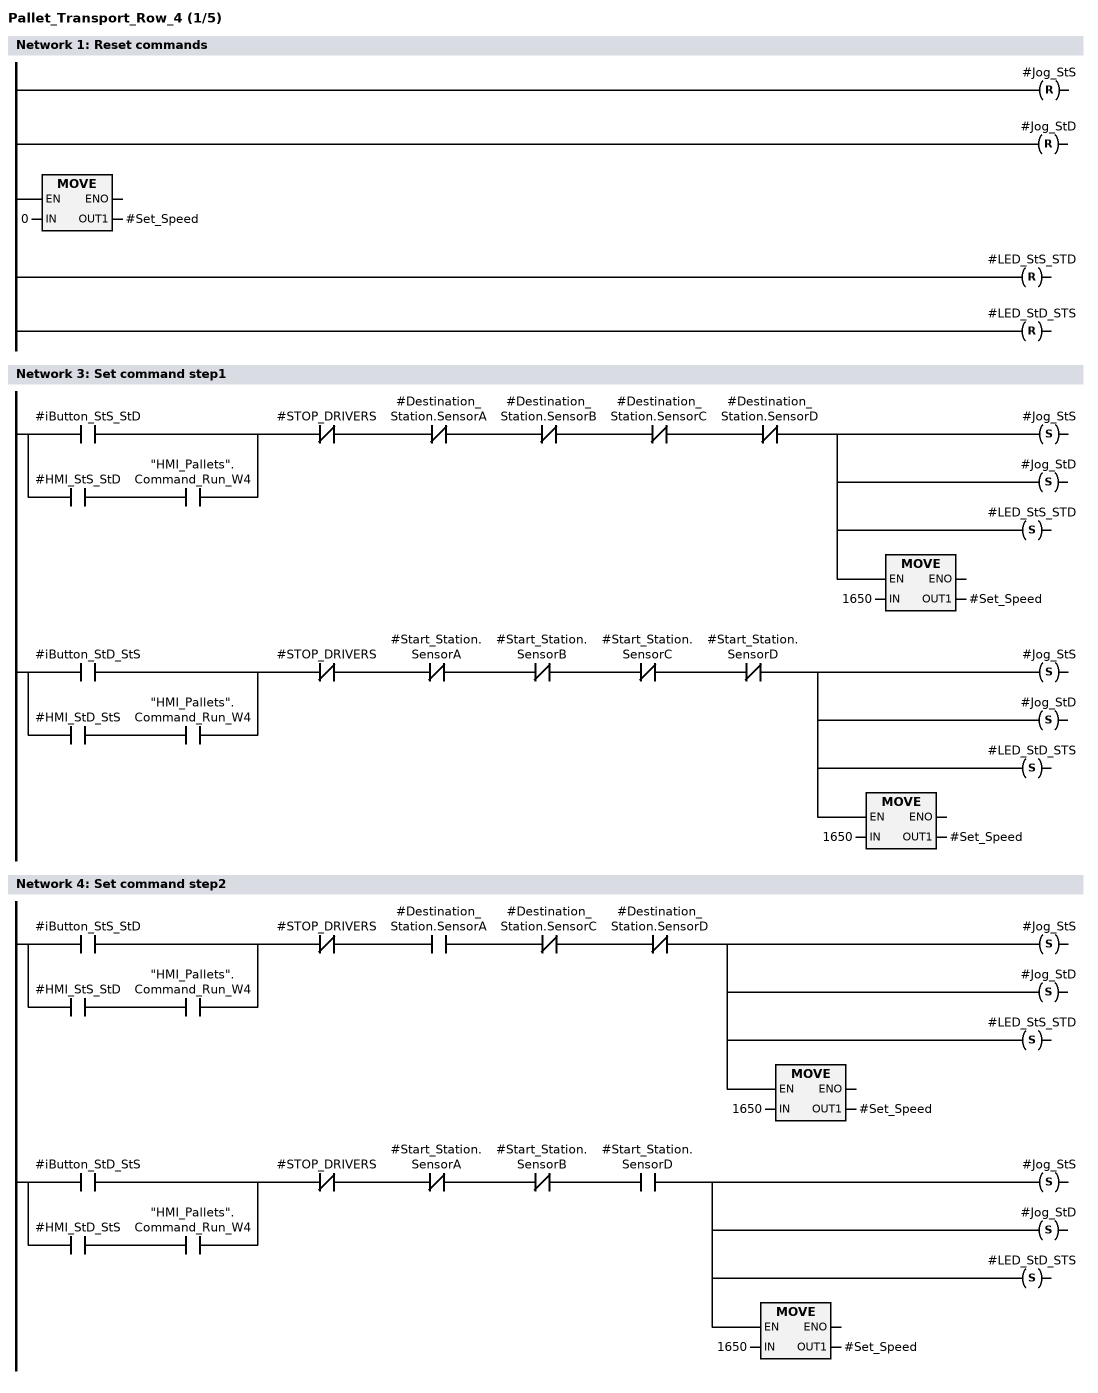
   RUNG wire#powerrail
      R_Coil( #Jog_StS )
   END_RUNG
   RUNG wire#powerrail
      R_Coil( #Jog_StD )
   END_RUNG
   RUNG wire#powerrail
      Move(in := 0, out1 => #Set_Speed)
   END_RUNG
   RUNG wire#powerrail
      R_Coil( #LED_StS_STD )
   END_RUNG
   RUNG wire#powerrail
      R_Coil( #LED_StD_STS )
   END_RUNG
   // the same network as SCL:
   #Jog_StS := FALSE;
   #Jog_StD := FALSE;
   #Set_Speed := 0;
   #LED_StS_STD := FALSE;
   #LED_StD_STS := FALSE;
END_REGION

REGION Network 2 (SCL): Triggers STOP_DRIVERS after 8 s of active move command without motion
   #Timer_Drive_Error_Button(
                             IN :=
                             (
                             #iButton_StS_StD OR
                             #iButton_StD_StS
                             )
                             AND NOT (
                             #oDriveStS_Param.x_Bit_4_Motor_turning OR
                             #oDriveStS_double_Param.x_Bit_4_Motor_turning OR
                             #oDriveStD_Param.x_Bit_4_Motor_turning OR
                             #oDriveStD_double_Param.x_Bit_4_Motor_turning
                             ),
                             PT := T#15s
   );


   #Timer_Drive_Error_HMI(
                          IN :=
                          (
                          #HMI_StS_StD OR
                          #HMI_StD_StS
                          )
                          AND NOT (
                          #oDriveStS_Param.x_Bit_4_Motor_turning OR
                          #oDriveStS_double_Param.x_Bit_4_Motor_turning OR
                          #oDriveStD_Param.x_Bit_4_Motor_turning OR
                          #oDriveStD_double_Param.x_Bit_4_Motor_turning
                          ),
                          PT := T#10s
   );

   IF #Timer_Drive_Error_Button.Q THEN
       #STOP_DRIVERS := TRUE;
       #Stop_Drive_Button := TRUE;
   END_IF;


   IF #Timer_Drive_Error_HMI.Q THEN
       #STOP_DRIVERS := TRUE;
       #Stop_Drive_HMI := TRUE;
       #HMI_StS_StD := FALSE;
       #HMI_StD_StS := FALSE;
   END_IF;


   IF "HMI_Pallets".Reset_Drivers THEN
       #STOP_DRIVERS := FALSE;
       #Stop_Drive_Button := FALSE;
       #Stop_Drive_HMI := FALSE;
   END_IF;
END_REGION

REGION Network 3: Set command step1
   RUNG wire#powerrail
      Contact( #iButton_StS_StD )
      wire#w1
      I_Contact( #STOP_DRIVERS )
      I_Contact( #Destination_Station.SensorA )
      I_Contact( #Destination_Station.SensorB )
      I_Contact( #Destination_Station.SensorC )
      I_Contact( #Destination_Station.SensorD )
      wire#w2
      S_Coil( #Jog_StS )
   END_RUNG
   RUNG wire#powerrail
      Contact( #HMI_StS_StD )
      Contact( "HMI_Pallets".Command_Run_W4 )
   END_RUNG wire#w1
   RUNG wire#w2
      S_Coil( #Jog_StD )
   END_RUNG
   RUNG wire#w2
      S_Coil( #LED_StS_STD )
   END_RUNG
   RUNG wire#w2
      Move(in := 1650, out1 => #Set_Speed)
   END_RUNG
   RUNG wire#powerrail
      Contact( #iButton_StD_StS )
      wire#w3
      I_Contact( #STOP_DRIVERS )
      I_Contact( #Start_Station.SensorA )
      I_Contact( #Start_Station.SensorB )
      I_Contact( #Start_Station.SensorC )
      I_Contact( #Start_Station.SensorD )
      wire#w4
      S_Coil( #Jog_StS )
   END_RUNG
   RUNG wire#powerrail
      Contact( #HMI_StD_StS )
      Contact( "HMI_Pallets".Command_Run_W4 )
   END_RUNG wire#w3
   RUNG wire#w4
      S_Coil( #Jog_StD )
   END_RUNG
   RUNG wire#w4
      S_Coil( #LED_StD_STS )
   END_RUNG
   RUNG wire#w4
      Move(in := 1650, out1 => #Set_Speed)
   END_RUNG
   // the same network as SCL:
   IF (#iButton_StS_StD OR (#HMI_StS_StD AND "HMI_Pallets".Command_Run_W4)) AND NOT #STOP_DRIVERS AND NOT #Destination_Station.SensorA AND NOT #Destination_Station.SensorB AND NOT #Destination_Station.SensorC AND NOT #Destination_Station.SensorD THEN
       #Jog_StS := TRUE;
       #Jog_StD := TRUE;
       #LED_StS_STD := TRUE;
       #Set_Speed := 1650;
   END_IF;
   IF (#iButton_StD_StS OR (#HMI_StD_StS AND "HMI_Pallets".Command_Run_W4)) AND NOT #STOP_DRIVERS AND NOT #Start_Station.SensorA AND NOT #Start_Station.SensorB AND NOT #Start_Station.SensorC AND NOT #Start_Station.SensorD THEN
       #Jog_StS := TRUE;
       #Jog_StD := TRUE;
       #LED_StD_STS := TRUE;
       #Set_Speed := 1650;
   END_IF;
END_REGION

REGION Network 4: Set command step2
   RUNG wire#powerrail
      Contact( #iButton_StS_StD )
      wire#w1
      I_Contact( #STOP_DRIVERS )
      Contact( #Destination_Station.SensorA )
      I_Contact( #Destination_Station.SensorC )
      I_Contact( #Destination_Station.SensorD )
      wire#w2
      S_Coil( #Jog_StS )
   END_RUNG
   RUNG wire#powerrail
      Contact( #HMI_StS_StD )
      Contact( "HMI_Pallets".Command_Run_W4 )
   END_RUNG wire#w1
   RUNG wire#w2
      S_Coil( #Jog_StD )
   END_RUNG
   RUNG wire#w2
      S_Coil( #LED_StS_STD )
   END_RUNG
   RUNG wire#w2
      Move(in := 1650, out1 => #Set_Speed)
   END_RUNG
   RUNG wire#powerrail
      Contact( #iButton_StD_StS )
      wire#w3
      I_Contact( #STOP_DRIVERS )
      I_Contact( #Start_Station.SensorA )
      I_Contact( #Start_Station.SensorB )
      Contact( #Start_Station.SensorD )
      wire#w4
      S_Coil( #Jog_StS )
   END_RUNG
   RUNG wire#powerrail
      Contact( #HMI_StD_StS )
      Contact( "HMI_Pallets".Command_Run_W4 )
   END_RUNG wire#w3
   RUNG wire#w4
      S_Coil( #Jog_StD )
   END_RUNG
   RUNG wire#w4
      S_Coil( #LED_StD_STS )
   END_RUNG
   RUNG wire#w4
      Move(in := 1650, out1 => #Set_Speed)
   END_RUNG
   // the same network as SCL:
   IF (#iButton_StS_StD OR (#HMI_StS_StD AND "HMI_Pallets".Command_Run_W4)) AND NOT #STOP_DRIVERS AND #Destination_Station.SensorA AND NOT #Destination_Station.SensorC AND NOT #Destination_Station.SensorD THEN
       #Jog_StS := TRUE;
       #Jog_StD := TRUE;
       #LED_StS_STD := TRUE;
       #Set_Speed := 1650;
   END_IF;
   IF (#iButton_StD_StS OR (#HMI_StD_StS AND "HMI_Pallets".Command_Run_W4)) AND NOT #STOP_DRIVERS AND NOT #Start_Station.SensorA AND NOT #Start_Station.SensorB AND #Start_Station.SensorD THEN
       #Jog_StS := TRUE;
       #Jog_StD := TRUE;
       #LED_StD_STS := TRUE;
       #Set_Speed := 1650;
   END_IF;
END_REGION

REGION Network 5: Set command step3
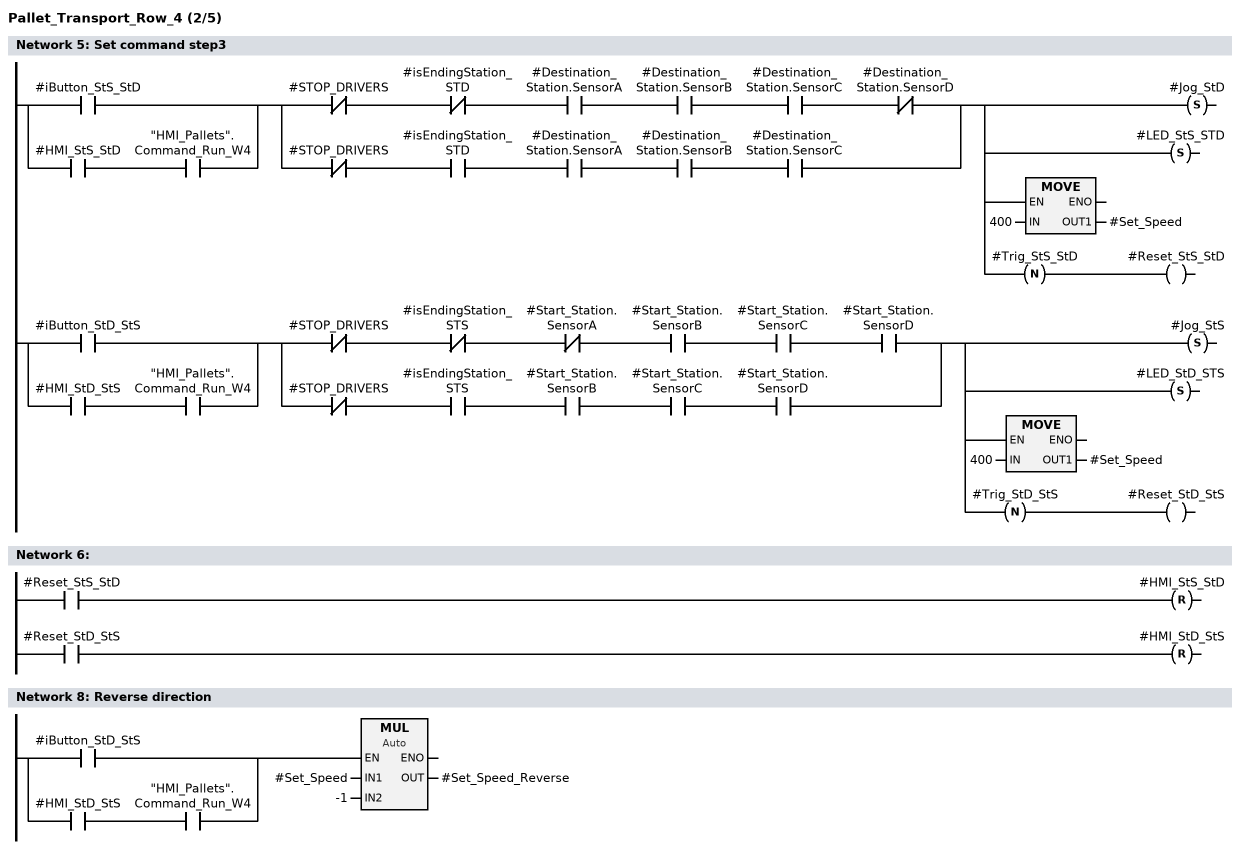
   RUNG wire#powerrail
      Contact( #iButton_StS_StD )
      wire#w1
      I_Contact( #STOP_DRIVERS )
      I_Contact( #isEndingStation_STD )
      Contact( #Destination_Station.SensorA )
      Contact( #Destination_Station.SensorB )
      Contact( #Destination_Station.SensorC )
      I_Contact( #Destination_Station.SensorD )
      wire#w2
      S_Coil( #Jog_StD )
   END_RUNG
   RUNG wire#powerrail
      Contact( #HMI_StS_StD )
      Contact( "HMI_Pallets".Command_Run_W4 )
   END_RUNG wire#w1
   RUNG wire#w1
      I_Contact( #STOP_DRIVERS )
      Contact( #isEndingStation_STD )
      Contact( #Destination_Station.SensorA )
      Contact( #Destination_Station.SensorB )
      Contact( #Destination_Station.SensorC )
   END_RUNG wire#w2
   RUNG wire#w2
      S_Coil( #LED_StS_STD )
   END_RUNG
   RUNG wire#w2
      Move(in := 400, out1 => #Set_Speed)
   END_RUNG
   RUNG wire#w2
      N_Trig( #Trig_StS_StD )
      Coil( #Reset_StS_StD )
   END_RUNG
   RUNG wire#powerrail
      Contact( #iButton_StD_StS )
      wire#w3
      I_Contact( #STOP_DRIVERS )
      I_Contact( #isEndingStation_STS )
      I_Contact( #Start_Station.SensorA )
      Contact( #Start_Station.SensorB )
      Contact( #Start_Station.SensorC )
      Contact( #Start_Station.SensorD )
      wire#w4
      S_Coil( #Jog_StS )
   END_RUNG
   RUNG wire#powerrail
      Contact( #HMI_StD_StS )
      Contact( "HMI_Pallets".Command_Run_W4 )
   END_RUNG wire#w3
   RUNG wire#w3
      I_Contact( #STOP_DRIVERS )
      Contact( #isEndingStation_STS )
      Contact( #Start_Station.SensorB )
      Contact( #Start_Station.SensorC )
      Contact( #Start_Station.SensorD )
   END_RUNG wire#w4
   RUNG wire#w4
      S_Coil( #LED_StD_STS )
   END_RUNG
   RUNG wire#w4
      Move(in := 400, out1 => #Set_Speed)
   END_RUNG
   RUNG wire#w4
      N_Trig( #Trig_StD_StS )
      Coil( #Reset_StD_StS )
   END_RUNG
   // the same network as SCL:
   #_w1 := (#iButton_StS_StD OR (#HMI_StS_StD AND "HMI_Pallets".Command_Run_W4)) AND ((NOT #STOP_DRIVERS AND NOT #isEndingStation_STD AND #Destination_Station.SensorA AND #Destination_Station.SensorB AND #Destination_Station.SensorC AND NOT #Destination_Station.SensorD) OR (NOT #STOP_DRIVERS AND #isEndingStation_STD AND #Destination_Station.SensorA AND #Destination_Station.SensorB AND #Destination_Station.SensorC));
   IF #_w1 THEN
       #Jog_StD := TRUE;
       #LED_StS_STD := TRUE;
       #Set_Speed := 400;
   END_IF;
   #_w2 := NOT #_w1 AND #Trig_StS_StD;   // falling edge
   #Trig_StS_StD := #_w1;
   #Reset_StS_StD := #_w2;
   #_w3 := (#iButton_StD_StS OR (#HMI_StD_StS AND "HMI_Pallets".Command_Run_W4)) AND ((NOT #STOP_DRIVERS AND NOT #isEndingStation_STS AND NOT #Start_Station.SensorA AND #Start_Station.SensorB AND #Start_Station.SensorC AND #Start_Station.SensorD) OR (NOT #STOP_DRIVERS AND #isEndingStation_STS AND #Start_Station.SensorB AND #Start_Station.SensorC AND #Start_Station.SensorD));
   IF #_w3 THEN
       #Jog_StS := TRUE;
       #LED_StD_STS := TRUE;
       #Set_Speed := 400;
   END_IF;
   #_w4 := NOT #_w3 AND #Trig_StD_StS;   // falling edge
   #Trig_StD_StS := #_w3;
   #Reset_StD_StS := #_w4;
END_REGION

REGION Network 6
   RUNG wire#powerrail
      Contact( #Reset_StS_StD )
      R_Coil( #HMI_StS_StD )
   END_RUNG
   RUNG wire#powerrail
      Contact( #Reset_StD_StS )
      R_Coil( #HMI_StD_StS )
   END_RUNG
   // the same network as SCL:
   IF #Reset_StS_StD THEN #HMI_StS_StD := FALSE; END_IF;
   IF #Reset_StD_StS THEN #HMI_StD_StS := FALSE; END_IF;
END_REGION

REGION Network 7 (SCL): Centering
   IF NOT #Destination_Station.SensorB OR
       NOT #Destination_Station.SensorC THEN
       #oCentering := 0;
       #CenteringStep := 0;
       IF #isCentering THEN
           #Centering_Alarm := TRUE;
           #isCentering := FALSE;
       END_IF;
   END_IF;

   IF #isCentering THEN
       CASE #CenteringStep OF
           0:
               IF #Destination_Station.SensorB AND
                   #Destination_Station.SensorC AND
                   #Destination_Station.SensorD THEN
                   #Set_Speed := #SPEED_BACK;
                   //#Jog_StS := TRUE;
                   #Jog_StD := TRUE;
               END_IF;

               IF  #Destination_Station.SensorB AND
                   #Destination_Station.SensorC AND
                   NOT #Destination_Station.SensorD THEN
                   #CenteringStep := 1;
               END_IF;

           1:
               #Set_Speed := #SPEED_FWD;
               //  #Jog_StS := TRUE;
               #Jog_StD := TRUE;
               IF #Destination_Station.SensorD THEN
                   #CenteringStep := 2;
               END_IF;

           2:
               #Set_Speed := 0;
               // #Jog_StS := FALSE;
               #Jog_StD := FALSE;
               #oCentering := TRUE;
               #CenteringStep := 0;
               #isCentering := FALSE;
               #Centering_Alarm := FALSE;
       END_CASE;
   END_IF;

   #TON_Centering(IN := #isCentering,
                  PT := T#8s);

   #trigTimeout(CLK := #TON_Centering.Q);

   // Wykona się tylko raz, gdy minie 8s
   IF #trigTimeout.Q THEN
       #Centering_Alarm := TRUE;
       #isCentering := FALSE;
       #CenteringStep := 0;
       #Set_Speed := 0;
       #Jog_StD := FALSE;
       #Jog_StS := FALSE;
   END_IF;
END_REGION

REGION Network 8: Reverse direction
   RUNG wire#powerrail
      Contact( #iButton_StD_StS )
      wire#w1
      Mul(in1 := #Set_Speed, in2 := -1, out => #Set_Speed_Reverse)
   END_RUNG
   RUNG wire#powerrail
      Contact( #HMI_StD_StS )
      Contact( "HMI_Pallets".Command_Run_W4 )
   END_RUNG wire#w1
   // the same network as SCL:
   IF #iButton_StD_StS OR (#HMI_StD_StS AND "HMI_Pallets".Command_Run_W4) THEN
       #Set_Speed_Reverse := #Set_Speed * (-1);
   END_IF;
END_REGION

REGION Network 9: StS Drive
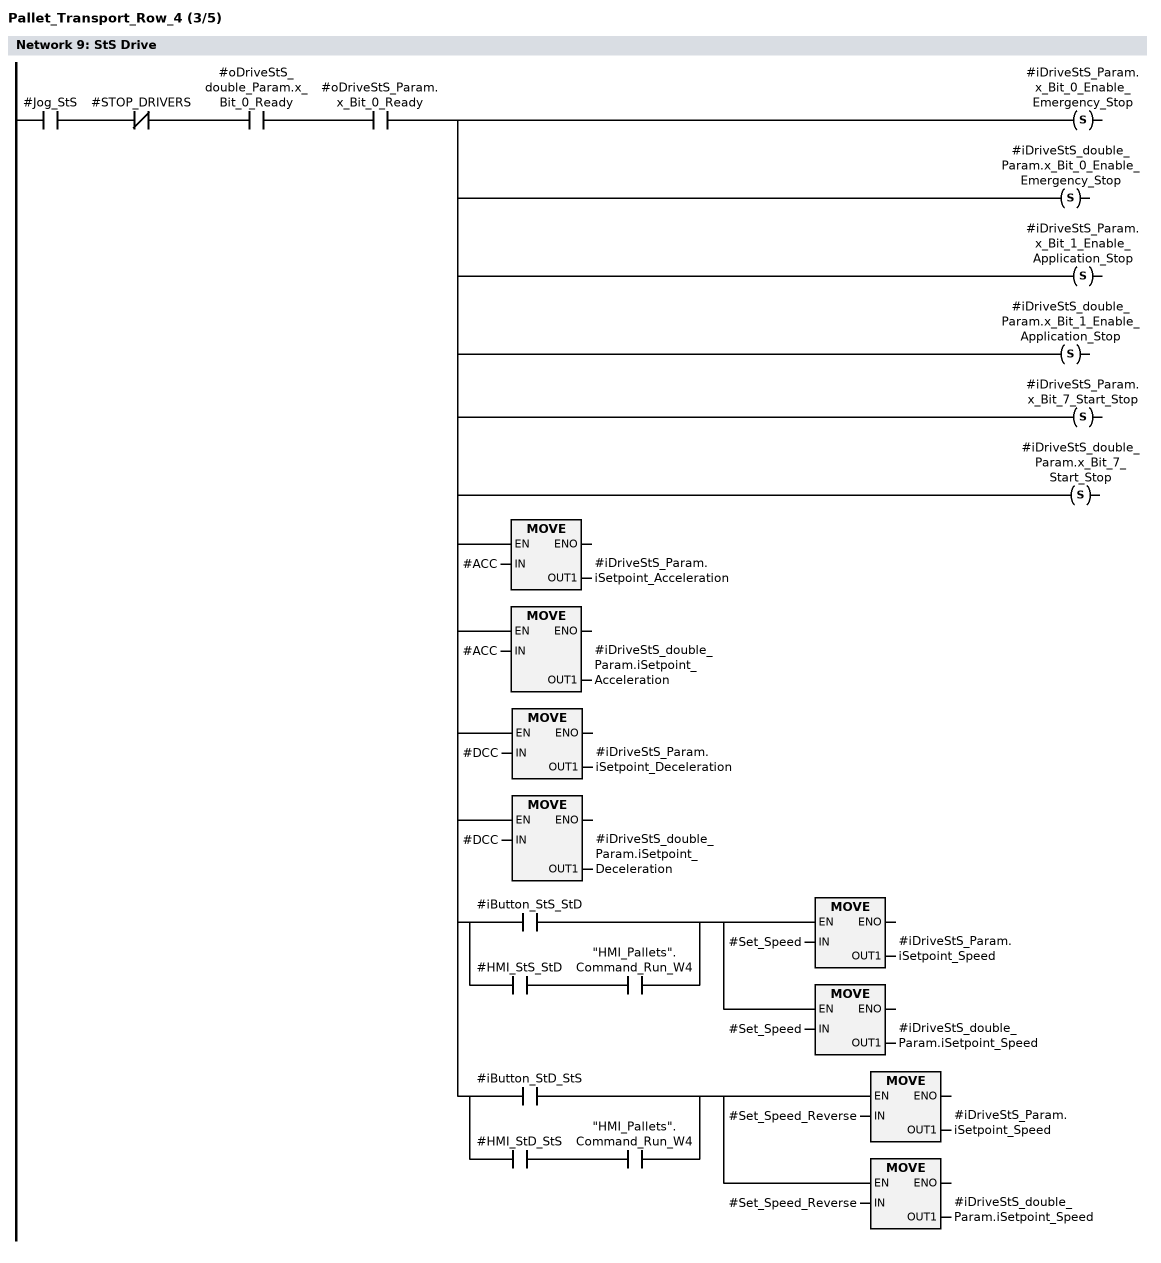
   RUNG wire#powerrail
      Contact( #Jog_StS )
      I_Contact( #STOP_DRIVERS )
      Contact( #oDriveStS_double_Param.x_Bit_0_Ready )
      Contact( #oDriveStS_Param.x_Bit_0_Ready )
      wire#w1
      S_Coil( #iDriveStS_Param.x_Bit_0_Enable_Emergency_Stop )
   END_RUNG
   RUNG wire#w1
      S_Coil( #iDriveStS_double_Param.x_Bit_0_Enable_Emergency_Stop )
   END_RUNG
   RUNG wire#w1
      S_Coil( #iDriveStS_Param.x_Bit_1_Enable_Application_Stop )
   END_RUNG
   RUNG wire#w1
      S_Coil( #iDriveStS_double_Param.x_Bit_1_Enable_Application_Stop )
   END_RUNG
   RUNG wire#w1
      S_Coil( #iDriveStS_Param.x_Bit_7_Start_Stop )
   END_RUNG
   RUNG wire#w1
      S_Coil( #iDriveStS_double_Param.x_Bit_7_Start_Stop )
   END_RUNG
   RUNG wire#w1
      Move(in := #ACC, out1 => #iDriveStS_Param.iSetpoint_Acceleration)
   END_RUNG
   RUNG wire#w1
      Move(in := #ACC, out1 => #iDriveStS_double_Param.iSetpoint_Acceleration)
   END_RUNG
   RUNG wire#w1
      Move(in := #DCC, out1 => #iDriveStS_Param.iSetpoint_Deceleration)
   END_RUNG
   RUNG wire#w1
      Move(in := #DCC, out1 => #iDriveStS_double_Param.iSetpoint_Deceleration)
   END_RUNG
   RUNG wire#w1
      Contact( #iButton_StS_StD )
      wire#w2
      Move(in := #Set_Speed, out1 => #iDriveStS_Param.iSetpoint_Speed)
   END_RUNG
   RUNG wire#w1
      Contact( #HMI_StS_StD )
      Contact( "HMI_Pallets".Command_Run_W4 )
   END_RUNG wire#w2
   RUNG wire#w2
      Move(in := #Set_Speed, out1 => #iDriveStS_double_Param.iSetpoint_Speed)
   END_RUNG
   RUNG wire#w1
      Contact( #iButton_StD_StS )
      wire#w3
      Move(in := #Set_Speed_Reverse, out1 => #iDriveStS_Param.iSetpoint_Speed)
   END_RUNG
   RUNG wire#w1
      Contact( #HMI_StD_StS )
      Contact( "HMI_Pallets".Command_Run_W4 )
   END_RUNG wire#w3
   RUNG wire#w3
      Move(in := #Set_Speed_Reverse, out1 => #iDriveStS_double_Param.iSetpoint_Speed)
   END_RUNG
   // the same network as SCL:
   #_w1 := #Jog_StS AND NOT #STOP_DRIVERS AND #oDriveStS_double_Param.x_Bit_0_Ready AND #oDriveStS_Param.x_Bit_0_Ready;
   IF #_w1 THEN
       #iDriveStS_Param.x_Bit_0_Enable_Emergency_Stop := TRUE;
       #iDriveStS_double_Param.x_Bit_0_Enable_Emergency_Stop := TRUE;
       #iDriveStS_Param.x_Bit_1_Enable_Application_Stop := TRUE;
       #iDriveStS_double_Param.x_Bit_1_Enable_Application_Stop := TRUE;
       #iDriveStS_Param.x_Bit_7_Start_Stop := TRUE;
       #iDriveStS_double_Param.x_Bit_7_Start_Stop := TRUE;
       #iDriveStS_Param.iSetpoint_Acceleration := #ACC;
       #iDriveStS_double_Param.iSetpoint_Acceleration := #ACC;
       #iDriveStS_Param.iSetpoint_Deceleration := #DCC;
       #iDriveStS_double_Param.iSetpoint_Deceleration := #DCC;
   END_IF;
   IF #_w1 AND (#iButton_StS_StD OR (#HMI_StS_StD AND "HMI_Pallets".Command_Run_W4)) THEN
       #iDriveStS_Param.iSetpoint_Speed := #Set_Speed;
       #iDriveStS_double_Param.iSetpoint_Speed := #Set_Speed;
   END_IF;
   IF #_w1 AND (#iButton_StD_StS OR (#HMI_StD_StS AND "HMI_Pallets".Command_Run_W4)) THEN
       #iDriveStS_Param.iSetpoint_Speed := #Set_Speed_Reverse;
       #iDriveStS_double_Param.iSetpoint_Speed := #Set_Speed_Reverse;
   END_IF;
END_REGION

REGION Network 10: StC Drive
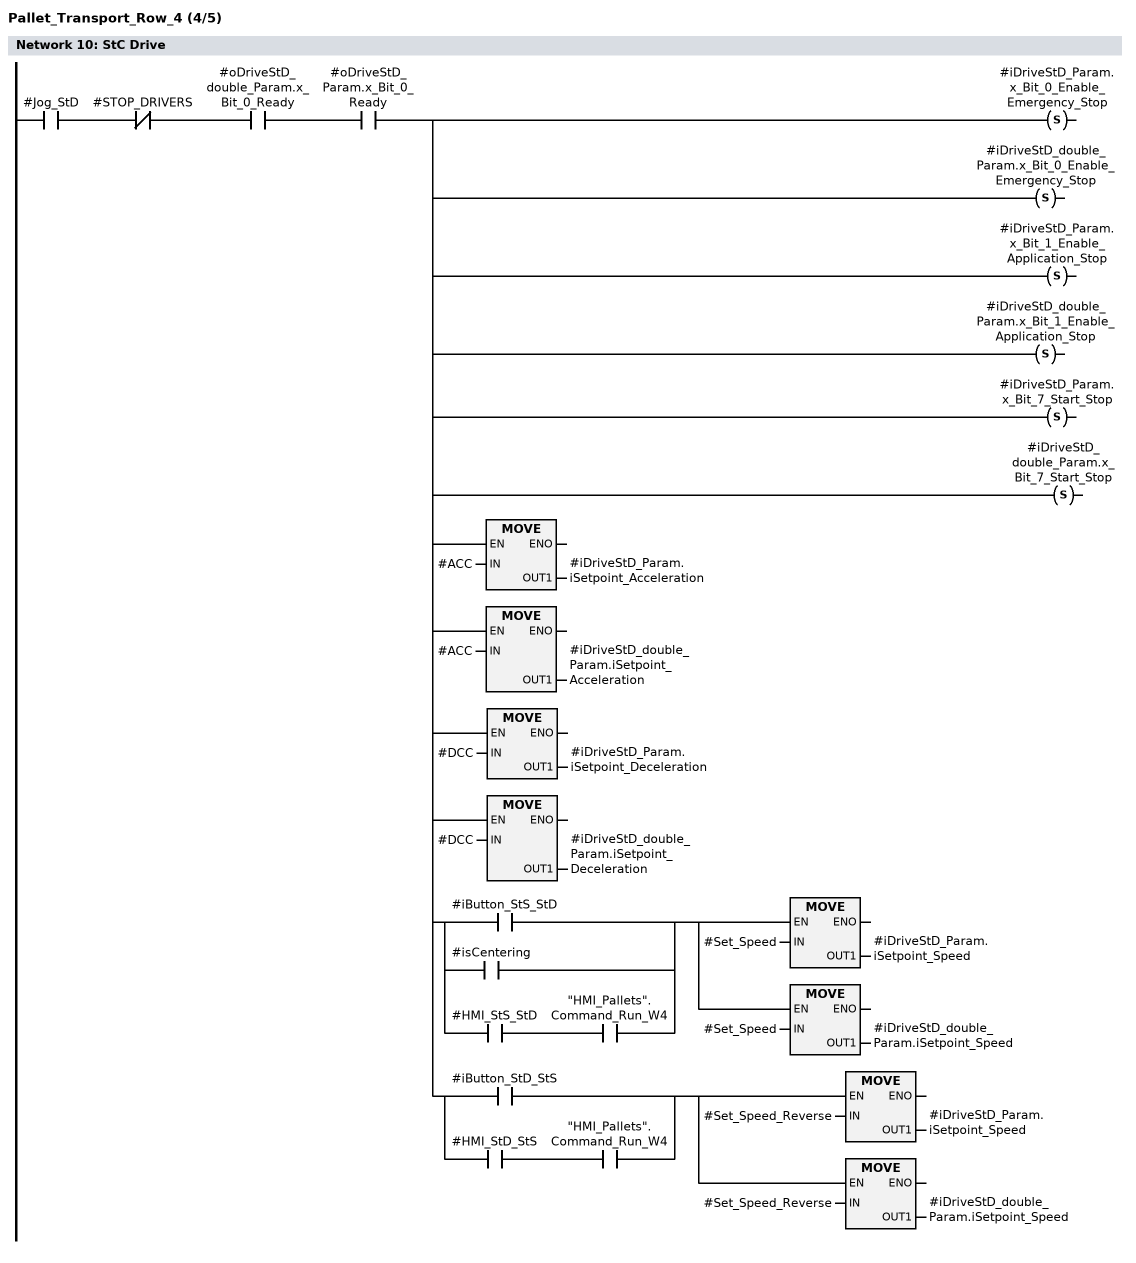
   RUNG wire#powerrail
      Contact( #Jog_StD )
      I_Contact( #STOP_DRIVERS )
      Contact( #oDriveStD_double_Param.x_Bit_0_Ready )
      Contact( #oDriveStD_Param.x_Bit_0_Ready )
      wire#w1
      S_Coil( #iDriveStD_Param.x_Bit_0_Enable_Emergency_Stop )
   END_RUNG
   RUNG wire#w1
      S_Coil( #iDriveStD_double_Param.x_Bit_0_Enable_Emergency_Stop )
   END_RUNG
   RUNG wire#w1
      S_Coil( #iDriveStD_Param.x_Bit_1_Enable_Application_Stop )
   END_RUNG
   RUNG wire#w1
      S_Coil( #iDriveStD_double_Param.x_Bit_1_Enable_Application_Stop )
   END_RUNG
   RUNG wire#w1
      S_Coil( #iDriveStD_Param.x_Bit_7_Start_Stop )
   END_RUNG
   RUNG wire#w1
      S_Coil( #iDriveStD_double_Param.x_Bit_7_Start_Stop )
   END_RUNG
   RUNG wire#w1
      Move(in := #ACC, out1 => #iDriveStD_Param.iSetpoint_Acceleration)
   END_RUNG
   RUNG wire#w1
      Move(in := #ACC, out1 => #iDriveStD_double_Param.iSetpoint_Acceleration)
   END_RUNG
   RUNG wire#w1
      Move(in := #DCC, out1 => #iDriveStD_Param.iSetpoint_Deceleration)
   END_RUNG
   RUNG wire#w1
      Move(in := #DCC, out1 => #iDriveStD_double_Param.iSetpoint_Deceleration)
   END_RUNG
   RUNG wire#w1
      Contact( #iButton_StS_StD )
      wire#w2
      Move(in := #Set_Speed, out1 => #iDriveStD_Param.iSetpoint_Speed)
   END_RUNG
   RUNG wire#w1
      Contact( #isCentering )
   END_RUNG wire#w2
   RUNG wire#w1
      Contact( #HMI_StS_StD )
      Contact( "HMI_Pallets".Command_Run_W4 )
   END_RUNG wire#w2
   RUNG wire#w2
      Move(in := #Set_Speed, out1 => #iDriveStD_double_Param.iSetpoint_Speed)
   END_RUNG
   RUNG wire#w1
      Contact( #iButton_StD_StS )
      wire#w3
      Move(in := #Set_Speed_Reverse, out1 => #iDriveStD_Param.iSetpoint_Speed)
   END_RUNG
   RUNG wire#w1
      Contact( #HMI_StD_StS )
      Contact( "HMI_Pallets".Command_Run_W4 )
   END_RUNG wire#w3
   RUNG wire#w3
      Move(in := #Set_Speed_Reverse, out1 => #iDriveStD_double_Param.iSetpoint_Speed)
   END_RUNG
   // the same network as SCL:
   #_w1 := #Jog_StD AND NOT #STOP_DRIVERS AND #oDriveStD_double_Param.x_Bit_0_Ready AND #oDriveStD_Param.x_Bit_0_Ready;
   IF #_w1 THEN
       #iDriveStD_Param.x_Bit_0_Enable_Emergency_Stop := TRUE;
       #iDriveStD_double_Param.x_Bit_0_Enable_Emergency_Stop := TRUE;
       #iDriveStD_Param.x_Bit_1_Enable_Application_Stop := TRUE;
       #iDriveStD_double_Param.x_Bit_1_Enable_Application_Stop := TRUE;
       #iDriveStD_Param.x_Bit_7_Start_Stop := TRUE;
       #iDriveStD_double_Param.x_Bit_7_Start_Stop := TRUE;
       #iDriveStD_Param.iSetpoint_Acceleration := #ACC;
       #iDriveStD_double_Param.iSetpoint_Acceleration := #ACC;
       #iDriveStD_Param.iSetpoint_Deceleration := #DCC;
       #iDriveStD_double_Param.iSetpoint_Deceleration := #DCC;
   END_IF;
   IF #_w1 AND (#iButton_StS_StD OR #isCentering OR (#HMI_StS_StD AND "HMI_Pallets".Command_Run_W4)) THEN
       #iDriveStD_Param.iSetpoint_Speed := #Set_Speed;
       #iDriveStD_double_Param.iSetpoint_Speed := #Set_Speed;
   END_IF;
   IF #_w1 AND (#iButton_StD_StS OR (#HMI_StD_StS AND "HMI_Pallets".Command_Run_W4)) THEN
       #iDriveStD_Param.iSetpoint_Speed := #Set_Speed_Reverse;
       #iDriveStD_double_Param.iSetpoint_Speed := #Set_Speed_Reverse;
   END_IF;
END_REGION

REGION Network 11: StS -> StD Status
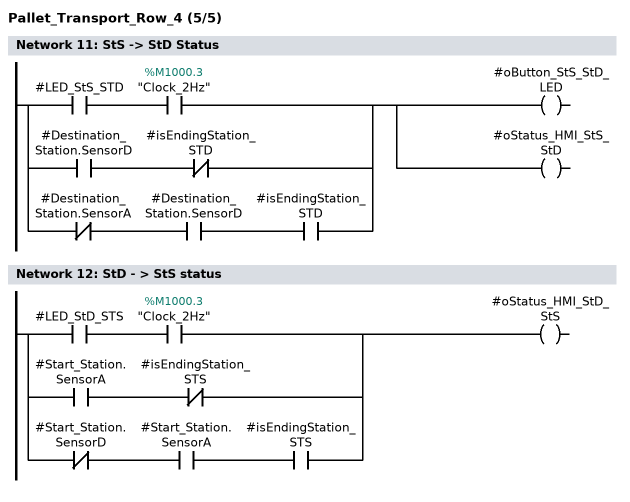
   RUNG wire#powerrail
      Contact( #LED_StS_STD )
      Contact( "Clock_2Hz" )
      wire#w1
      Coil( #oButton_StS_StD_LED )
   END_RUNG
   RUNG wire#powerrail
      Contact( #Destination_Station.SensorD )
      I_Contact( #isEndingStation_STD )
   END_RUNG wire#w1
   RUNG wire#powerrail
      I_Contact( #Destination_Station.SensorA )
      Contact( #Destination_Station.SensorD )
      Contact( #isEndingStation_STD )
   END_RUNG wire#w1
   RUNG wire#w1
      Coil( #oStatus_HMI_StS_StD )
   END_RUNG
   // the same network as SCL:
   #oButton_StS_StD_LED := (#LED_StS_STD AND "Clock_2Hz") OR (#Destination_Station.SensorD AND NOT #isEndingStation_STD) OR (NOT #Destination_Station.SensorA AND #Destination_Station.SensorD AND #isEndingStation_STD);
   #oStatus_HMI_StS_StD := #oButton_StS_StD_LED;
END_REGION

REGION Network 12: StD - > StS status
   RUNG wire#powerrail
      Contact( #LED_StD_STS )
      Contact( "Clock_2Hz" )
      wire#w1
      Coil( #oStatus_HMI_StD_StS )
   END_RUNG
   RUNG wire#powerrail
      Contact( #Start_Station.SensorA )
      I_Contact( #isEndingStation_STS )
   END_RUNG wire#w1
   RUNG wire#powerrail
      I_Contact( #Start_Station.SensorD )
      Contact( #Start_Station.SensorA )
      Contact( #isEndingStation_STS )
   END_RUNG wire#w1
   // the same network as SCL:
   #oStatus_HMI_StD_StS := (#LED_StD_STS AND "Clock_2Hz") OR (#Start_Station.SensorA AND NOT #isEndingStation_STS) OR (NOT #Start_Station.SensorD AND #Start_Station.SensorA AND #isEndingStation_STS);
END_REGION

REGION Network 13 (SCL): Centering status reset
   IF #oCentering AND (#iDriveStD_Param.x_Bit_1_Enable_Application_Stop  OR NOT #Destination_Station.SensorD) THEN
       #oCentering := 0;
   END_IF;
END_REGION
END_FUNCTION_BLOCK

FUNCTION_BLOCK "Pallet_Transport_Row_1_2"   // FB16, LAD
{ S7_Optimized_Access := 'TRUE' }
// stored: MemoryReserve 100, SetENOAutomatically false
   VAR_INPUT
      Start_Station : "Station";
      Destination_Station : "Station";
      Reverse_Rotation : Bool;
      iButton_StS_StD : Bool;
      iButton_StD_StS : Bool;
      isEndingStation_STD : Bool;
      isEndingStation_STS : Bool;
      isTippler : Bool;
      CompactionPermition : Bool := true;
   END_VAR
   VAR_OUTPUT
      oButton_StS_StD_LED : Bool;
      oButton_StD_StS_LED : Bool;
      oHMI_status_StS_StD : Bool;
      oHMI_status_StD_StS : Bool;
      oCentering : Bool;
      Stop_Drive_Button : Bool;
      Stop_Drive_HMI : Bool;
      Centering_Alarm : Bool;
   END_VAR
   VAR_IN_OUT
      iDriveStS_Param : "SEW_MOVIKIT_VelocityDrive_SETPOINTS_V2.1";
      oDriveStS_Param : "SEW_MOVIKIT_VelocityDrive_STATUS_V2.1";
      iDriveStD_Param : "SEW_MOVIKIT_VelocityDrive_SETPOINTS_V2.1";
      oDriveStD_Param : "SEW_MOVIKIT_VelocityDrive_STATUS_V2.1";
      iDriveStS_double_Param : "SEW_MOVIKIT_VelocityDrive_SETPOINTS_V2.1";
      oDriveStS_double_Param : "SEW_MOVIKIT_VelocityDrive_STATUS_V2.1";
      iDriveStD_double_Param : "SEW_MOVIKIT_VelocityDrive_SETPOINTS_V2.1";
      oDriveStD_double_Param : "SEW_MOVIKIT_VelocityDrive_STATUS_V2.1";
      isCentering : Bool;
      HMI_StS_StD : Bool;
      HMI_StD_StS : Bool;
   END_VAR
   VAR
      Drive_To_Destination : Bool;
      Set_Speed : Int;
      Set_Speed_Reverse : Int;
      CommunicationOk : Bool;
      Jog_StS : Bool;
      Jog_StD : Bool;
      CenteringStep : Int;
      TON_Centering : TON_TIME;
      trigTimeout { S7_SetPoint := 'True'} : R_TRIG;
      Trig_StS_StD { S7_SetPoint := 'True'} : Bool;
      Trig_StD_StS : Bool;
      Reset_StS_StD : Bool;
      Reset_StD_StS : Bool;
      PalletStep2 : Bool;
      Pallet_Go_StS_StD : Bool;
      Pallet_Go_StD_StS : Bool;
      Timer_Drive_Error_HMI : TON_TIME;
      Timer_Drive_Error_Button : TON_TIME;
      STOP_DRIVERS : Bool;
   END_VAR
   VAR_TEMP
      LED_StS_STD : Bool;
      LED_StD_StS : Bool;
      i : SInt;
      FoundIndex : SInt;
   END_VAR
   VAR CONSTANT
      ACC : Int := 300;
      DCC : Int := 300;
      SPEED_BACK : Int := -100;
      SPEED_FWD : Int := 100;
   END_VAR
   // Timer_Drive_Error_HMI.PT := T#8s;
   // Timer_Drive_Error_Button.PT := T#8s;
   VAR_TEMP   // added for the SCL form of the ladder/FBD networks
      _w1 : Bool;
      _w2 : Bool;
      _w3 : Bool;
      _w4 : Bool;
   END_VAR
BEGIN

REGION Network 1: Reset commands
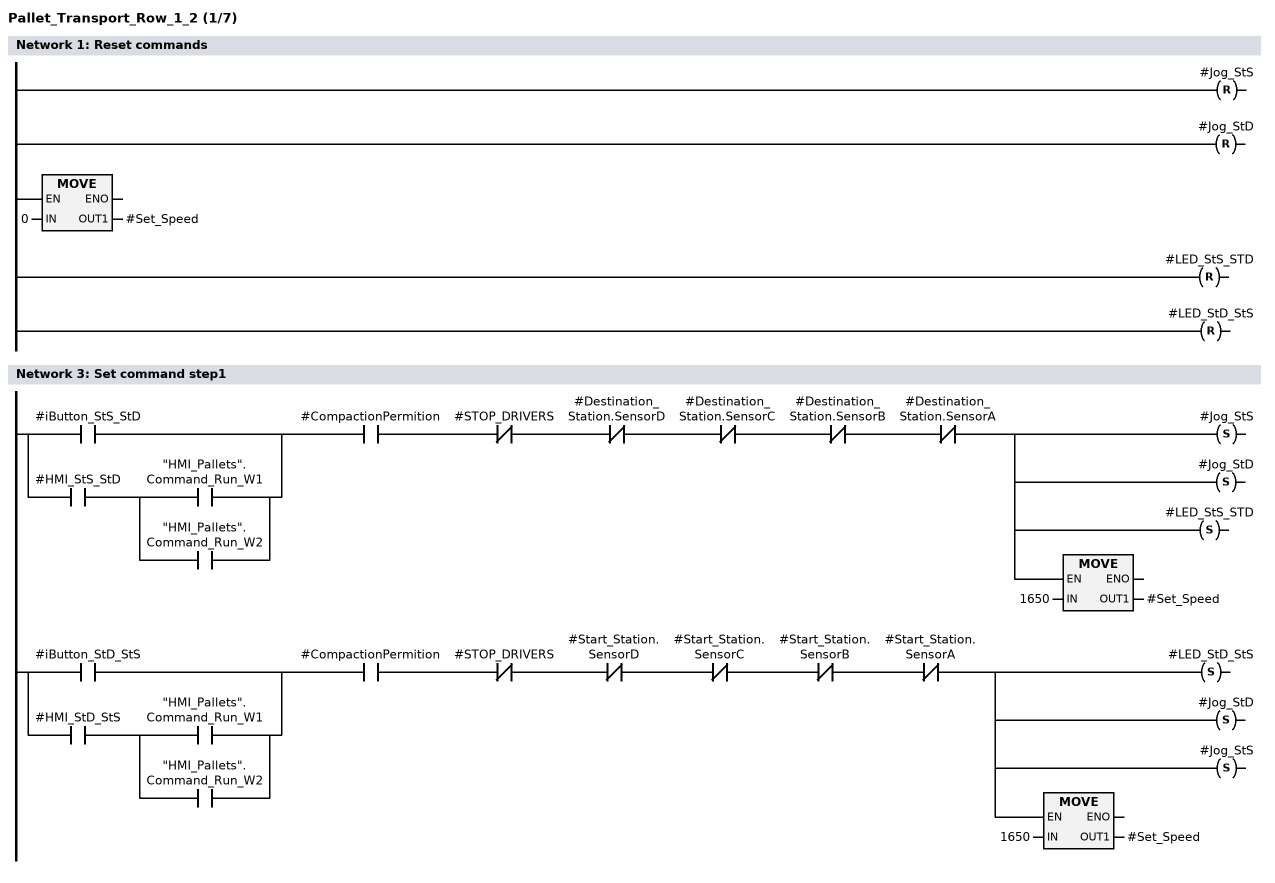
   RUNG wire#powerrail
      R_Coil( #Jog_StS )
   END_RUNG
   RUNG wire#powerrail
      R_Coil( #Jog_StD )
   END_RUNG
   RUNG wire#powerrail
      Move(in := 0, out1 => #Set_Speed)
   END_RUNG
   RUNG wire#powerrail
      R_Coil( #LED_StS_STD )
   END_RUNG
   RUNG wire#powerrail
      R_Coil( #LED_StD_StS )
   END_RUNG
   // the same network as SCL:
   #Jog_StS := FALSE;
   #Jog_StD := FALSE;
   #Set_Speed := 0;
   #LED_StS_STD := FALSE;
   #LED_StD_StS := FALSE;
END_REGION

REGION Network 2 (SCL): Triggers STOP_DRIVERS after 8 s of active move command without motion
   #Timer_Drive_Error_Button(
                             IN :=
                             (
                             #iButton_StS_StD OR
                             #iButton_StD_StS
                             )
                             AND NOT (
                             #oDriveStS_Param.x_Bit_4_Motor_turning OR
                             #oDriveStS_double_Param.x_Bit_4_Motor_turning OR
                             #oDriveStD_Param.x_Bit_4_Motor_turning OR
                             #oDriveStD_double_Param.x_Bit_4_Motor_turning
                             ),
                             PT := T#15s
   );

   #Timer_Drive_Error_HMI(
                          IN :=
                          (
                          #HMI_StS_StD OR
                          #HMI_StD_StS
                          )
                          AND NOT (
                          #oDriveStS_Param.x_Bit_4_Motor_turning OR
                          #oDriveStS_double_Param.x_Bit_4_Motor_turning OR
                          #oDriveStD_Param.x_Bit_4_Motor_turning OR
                          #oDriveStD_double_Param.x_Bit_4_Motor_turning
                          ),
                          PT := T#10s
   );

   IF #Timer_Drive_Error_Button.Q THEN
       #STOP_DRIVERS := TRUE;
       #Stop_Drive_Button := TRUE;
   END_IF;

   IF #Timer_Drive_Error_HMI.Q THEN
       #STOP_DRIVERS := TRUE;
       #Stop_Drive_HMI := TRUE;
       #HMI_StS_StD := false;
       #HMI_StD_StS := false;
   END_IF;

   IF "HMI_Pallets".Reset_Drivers THEN
       #STOP_DRIVERS := FALSE;
       #Stop_Drive_Button := FALSE;
       #Stop_Drive_HMI := FALSE;
   END_IF;
END_REGION

REGION Network 3: Set command step1
   RUNG wire#powerrail
      Contact( #iButton_StS_StD )
      wire#w1
      Contact( #CompactionPermition )
      I_Contact( #STOP_DRIVERS )
      I_Contact( #Destination_Station.SensorD )
      I_Contact( #Destination_Station.SensorC )
      I_Contact( #Destination_Station.SensorB )
      I_Contact( #Destination_Station.SensorA )
      wire#w3
      S_Coil( #Jog_StS )
   END_RUNG
   RUNG wire#powerrail
      Contact( #HMI_StS_StD )
      wire#w2
      Contact( "HMI_Pallets".Command_Run_W1 )
   END_RUNG wire#w1
   RUNG wire#w2
      Contact( "HMI_Pallets".Command_Run_W2 )
   END_RUNG wire#w1
   RUNG wire#w3
      S_Coil( #Jog_StD )
   END_RUNG
   RUNG wire#w3
      S_Coil( #LED_StS_STD )
   END_RUNG
   RUNG wire#w3
      Move(in := 1650, out1 => #Set_Speed)
   END_RUNG
   RUNG wire#powerrail
      Contact( #iButton_StD_StS )
      wire#w4
      Contact( #CompactionPermition )
      I_Contact( #STOP_DRIVERS )
      I_Contact( #Start_Station.SensorD )
      I_Contact( #Start_Station.SensorC )
      I_Contact( #Start_Station.SensorB )
      I_Contact( #Start_Station.SensorA )
      wire#w6
      S_Coil( #LED_StD_StS )
   END_RUNG
   RUNG wire#powerrail
      Contact( #HMI_StD_StS )
      wire#w5
      Contact( "HMI_Pallets".Command_Run_W1 )
   END_RUNG wire#w4
   RUNG wire#w5
      Contact( "HMI_Pallets".Command_Run_W2 )
   END_RUNG wire#w4
   RUNG wire#w6
      S_Coil( #Jog_StD )
   END_RUNG
   RUNG wire#w6
      S_Coil( #Jog_StS )
   END_RUNG
   RUNG wire#w6
      Move(in := 1650, out1 => #Set_Speed)
   END_RUNG
   // the same network as SCL:
   IF (#iButton_StS_StD OR (#HMI_StS_StD AND ("HMI_Pallets".Command_Run_W1 OR "HMI_Pallets".Command_Run_W2))) AND #CompactionPermition AND NOT #STOP_DRIVERS AND NOT #Destination_Station.SensorD AND NOT #Destination_Station.SensorC AND NOT #Destination_Station.SensorB AND NOT #Destination_Station.SensorA THEN
       #Jog_StS := TRUE;
       #Jog_StD := TRUE;
       #LED_StS_STD := TRUE;
       #Set_Speed := 1650;
   END_IF;
   IF (#iButton_StD_StS OR (#HMI_StD_StS AND ("HMI_Pallets".Command_Run_W1 OR "HMI_Pallets".Command_Run_W2))) AND #CompactionPermition AND NOT #STOP_DRIVERS AND NOT #Start_Station.SensorD AND NOT #Start_Station.SensorC AND NOT #Start_Station.SensorB AND NOT #Start_Station.SensorA THEN
       #LED_StD_StS := TRUE;
       #Jog_StD := TRUE;
       #Jog_StS := TRUE;
       #Set_Speed := 1650;
   END_IF;
END_REGION

REGION Network 4: Set command step2
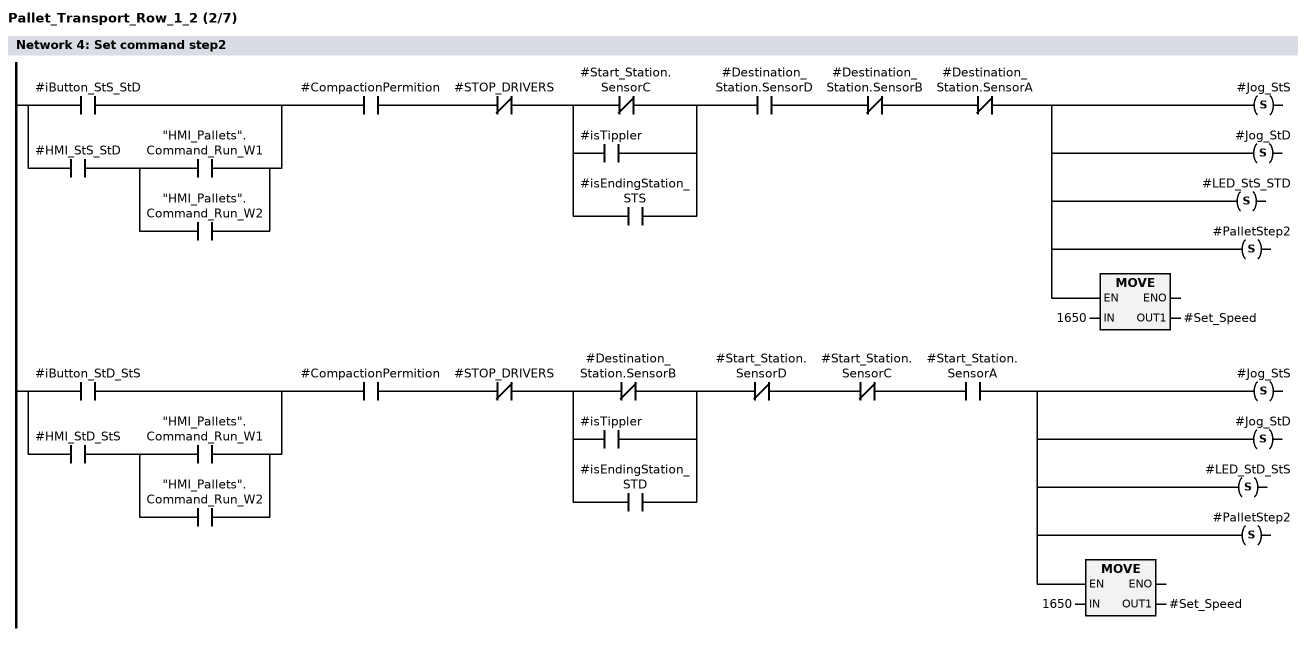
   RUNG wire#powerrail
      Contact( #iButton_StS_StD )
      wire#w1
      Contact( #CompactionPermition )
      I_Contact( #STOP_DRIVERS )
      wire#w3
      I_Contact( #Start_Station.SensorC )
      wire#w4
      Contact( #Destination_Station.SensorD )
      I_Contact( #Destination_Station.SensorB )
      I_Contact( #Destination_Station.SensorA )
      wire#w5
      S_Coil( #Jog_StS )
   END_RUNG
   RUNG wire#powerrail
      Contact( #HMI_StS_StD )
      wire#w2
      Contact( "HMI_Pallets".Command_Run_W1 )
   END_RUNG wire#w1
   RUNG wire#w2
      Contact( "HMI_Pallets".Command_Run_W2 )
   END_RUNG wire#w1
   RUNG wire#w3
      Contact( #isTippler )
   END_RUNG wire#w4
   RUNG wire#w3
      Contact( #isEndingStation_STS )
   END_RUNG wire#w4
   RUNG wire#w5
      S_Coil( #Jog_StD )
   END_RUNG
   RUNG wire#w5
      S_Coil( #LED_StS_STD )
   END_RUNG
   RUNG wire#w5
      S_Coil( #PalletStep2 )
   END_RUNG
   RUNG wire#w5
      Move(in := 1650, out1 => #Set_Speed)
   END_RUNG
   RUNG wire#powerrail
      Contact( #iButton_StD_StS )
      wire#w6
      Contact( #CompactionPermition )
      I_Contact( #STOP_DRIVERS )
      wire#w8
      I_Contact( #Destination_Station.SensorB )
      wire#w9
      I_Contact( #Start_Station.SensorD )
      I_Contact( #Start_Station.SensorC )
      Contact( #Start_Station.SensorA )
      wire#w10
      S_Coil( #Jog_StS )
   END_RUNG
   RUNG wire#powerrail
      Contact( #HMI_StD_StS )
      wire#w7
      Contact( "HMI_Pallets".Command_Run_W1 )
   END_RUNG wire#w6
   RUNG wire#w7
      Contact( "HMI_Pallets".Command_Run_W2 )
   END_RUNG wire#w6
   RUNG wire#w8
      Contact( #isTippler )
   END_RUNG wire#w9
   RUNG wire#w8
      Contact( #isEndingStation_STD )
   END_RUNG wire#w9
   RUNG wire#w10
      S_Coil( #Jog_StD )
   END_RUNG
   RUNG wire#w10
      S_Coil( #LED_StD_StS )
   END_RUNG
   RUNG wire#w10
      S_Coil( #PalletStep2 )
   END_RUNG
   RUNG wire#w10
      Move(in := 1650, out1 => #Set_Speed)
   END_RUNG
   // the same network as SCL:
   IF (#iButton_StS_StD OR (#HMI_StS_StD AND ("HMI_Pallets".Command_Run_W1 OR "HMI_Pallets".Command_Run_W2))) AND #CompactionPermition AND NOT #STOP_DRIVERS AND (NOT #Start_Station.SensorC OR #isTippler OR #isEndingStation_STS) AND #Destination_Station.SensorD AND NOT #Destination_Station.SensorB AND NOT #Destination_Station.SensorA THEN
       #Jog_StS := TRUE;
       #Jog_StD := TRUE;
       #LED_StS_STD := TRUE;
       #PalletStep2 := TRUE;
       #Set_Speed := 1650;
   END_IF;
   IF (#iButton_StD_StS OR (#HMI_StD_StS AND ("HMI_Pallets".Command_Run_W1 OR "HMI_Pallets".Command_Run_W2))) AND #CompactionPermition AND NOT #STOP_DRIVERS AND (NOT #Destination_Station.SensorB OR #isTippler OR #isEndingStation_STD) AND NOT #Start_Station.SensorD AND NOT #Start_Station.SensorC AND #Start_Station.SensorA THEN
       #Jog_StS := TRUE;
       #Jog_StD := TRUE;
       #LED_StD_StS := TRUE;
       #PalletStep2 := TRUE;
       #Set_Speed := 1650;
   END_IF;
END_REGION

REGION Network 5: Set command step3
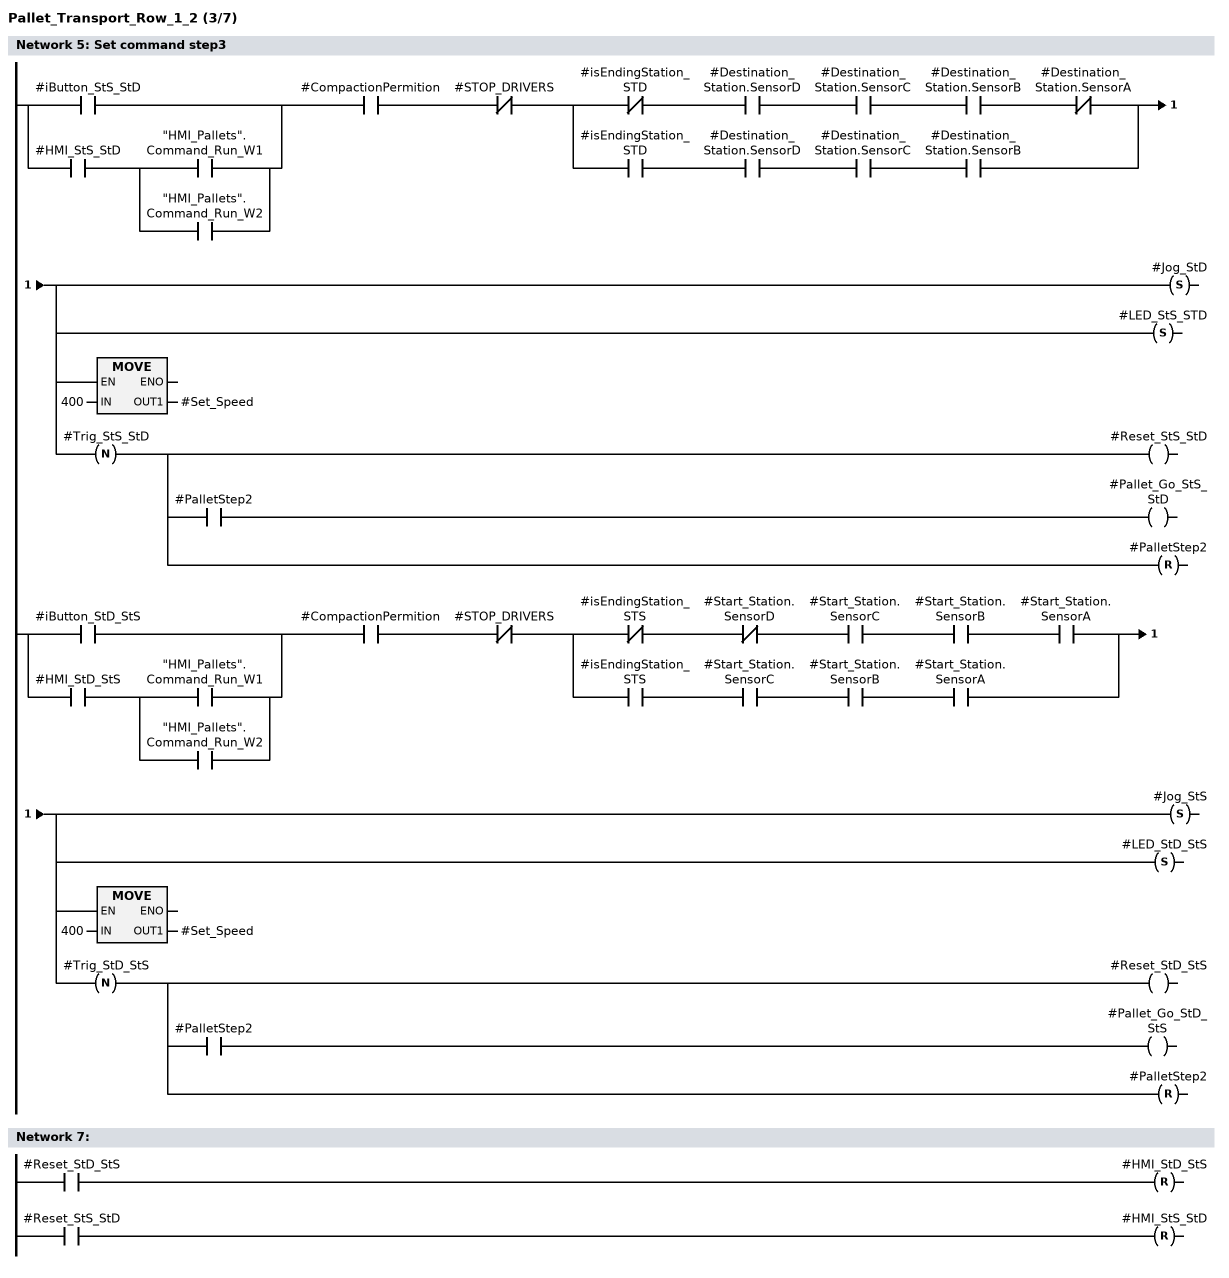
   RUNG wire#powerrail
      Contact( #iButton_StS_StD )
      wire#w1
      Contact( #CompactionPermition )
      I_Contact( #STOP_DRIVERS )
      wire#w3
      I_Contact( #isEndingStation_STD )
      Contact( #Destination_Station.SensorD )
      Contact( #Destination_Station.SensorC )
      Contact( #Destination_Station.SensorB )
      I_Contact( #Destination_Station.SensorA )
      wire#w4
      S_Coil( #Jog_StD )
   END_RUNG
   RUNG wire#powerrail
      Contact( #HMI_StS_StD )
      wire#w2
      Contact( "HMI_Pallets".Command_Run_W1 )
   END_RUNG wire#w1
   RUNG wire#w2
      Contact( "HMI_Pallets".Command_Run_W2 )
   END_RUNG wire#w1
   RUNG wire#w3
      Contact( #isEndingStation_STD )
      Contact( #Destination_Station.SensorD )
      Contact( #Destination_Station.SensorC )
      Contact( #Destination_Station.SensorB )
   END_RUNG wire#w4
   RUNG wire#w4
      S_Coil( #LED_StS_STD )
   END_RUNG
   RUNG wire#w4
      Move(in := 400, out1 => #Set_Speed)
   END_RUNG
   RUNG wire#w4
      N_Trig( #Trig_StS_StD )
      wire#w5
      Coil( #Reset_StS_StD )
   END_RUNG
   RUNG wire#w5
      Contact( #PalletStep2 )
      Coil( #Pallet_Go_StS_StD )
   END_RUNG
   RUNG wire#w5
      R_Coil( #PalletStep2 )
   END_RUNG
   RUNG wire#powerrail
      Contact( #iButton_StD_StS )
      wire#w6
      Contact( #CompactionPermition )
      I_Contact( #STOP_DRIVERS )
      wire#w8
      I_Contact( #isEndingStation_STS )
      I_Contact( #Start_Station.SensorD )
      Contact( #Start_Station.SensorC )
      Contact( #Start_Station.SensorB )
      Contact( #Start_Station.SensorA )
      wire#w9
      S_Coil( #Jog_StS )
   END_RUNG
   RUNG wire#powerrail
      Contact( #HMI_StD_StS )
      wire#w7
      Contact( "HMI_Pallets".Command_Run_W1 )
   END_RUNG wire#w6
   RUNG wire#w7
      Contact( "HMI_Pallets".Command_Run_W2 )
   END_RUNG wire#w6
   RUNG wire#w8
      Contact( #isEndingStation_STS )
      Contact( #Start_Station.SensorC )
      Contact( #Start_Station.SensorB )
      Contact( #Start_Station.SensorA )
   END_RUNG wire#w9
   RUNG wire#w9
      S_Coil( #LED_StD_StS )
   END_RUNG
   RUNG wire#w9
      Move(in := 400, out1 => #Set_Speed)
   END_RUNG
   RUNG wire#w9
      N_Trig( #Trig_StD_StS )
      wire#w10
      Coil( #Reset_StD_StS )
   END_RUNG
   RUNG wire#w10
      Contact( #PalletStep2 )
      Coil( #Pallet_Go_StD_StS )
   END_RUNG
   RUNG wire#w10
      R_Coil( #PalletStep2 )
   END_RUNG
   // the same network as SCL:
   #_w1 := (#iButton_StS_StD OR (#HMI_StS_StD AND ("HMI_Pallets".Command_Run_W1 OR "HMI_Pallets".Command_Run_W2))) AND #CompactionPermition AND NOT #STOP_DRIVERS AND ((NOT #isEndingStation_STD AND #Destination_Station.SensorD AND #Destination_Station.SensorC AND #Destination_Station.SensorB AND NOT #Destination_Station.SensorA) OR (#isEndingStation_STD AND #Destination_Station.SensorD AND #Destination_Station.SensorC AND #Destination_Station.SensorB));
   IF #_w1 THEN
       #Jog_StD := TRUE;
       #LED_StS_STD := TRUE;
       #Set_Speed := 400;
   END_IF;
   #_w2 := NOT #_w1 AND #Trig_StS_StD;   // falling edge
   #Trig_StS_StD := #_w1;
   #Reset_StS_StD := #_w2;
   #Pallet_Go_StS_StD := #_w2 AND #PalletStep2;
   IF #_w2 THEN #PalletStep2 := FALSE; END_IF;
   #_w3 := (#iButton_StD_StS OR (#HMI_StD_StS AND ("HMI_Pallets".Command_Run_W1 OR "HMI_Pallets".Command_Run_W2))) AND #CompactionPermition AND NOT #STOP_DRIVERS AND ((NOT #isEndingStation_STS AND NOT #Start_Station.SensorD AND #Start_Station.SensorC AND #Start_Station.SensorB AND #Start_Station.SensorA) OR (#isEndingStation_STS AND #Start_Station.SensorC AND #Start_Station.SensorB AND #Start_Station.SensorA));
   IF #_w3 THEN
       #Jog_StS := TRUE;
       #LED_StD_StS := TRUE;
       #Set_Speed := 400;
   END_IF;
   #_w4 := NOT #_w3 AND #Trig_StD_StS;   // falling edge
   #Trig_StD_StS := #_w3;
   #Reset_StD_StS := #_w4;
   #Pallet_Go_StD_StS := #_w4 AND #PalletStep2;
   IF #_w4 THEN #PalletStep2 := FALSE; END_IF;
END_REGION

REGION Network 6 (SCL): Move pallet in HMI system TODO
       #FoundIndex := 0;
       IF #Pallet_Go_StS_StD THEN
           FOR #i := 1 TO 24 DO
               IF ("Pallets_Stations".Pallets[#i].Station_Current_Position[2] = #Start_Station.Column) AND
                   ("Pallets_Stations".Pallets[#i].Station_Current_Position[1] = #Start_Station.Row) THEN
                   #FoundIndex := #i;
                   EXIT;
               END_IF;
           END_FOR;

       ELSIF #Pallet_Go_StD_StS THEN
           FOR #i := 1 TO 24 DO
               IF ("Pallets_Stations".Pallets[#i].Station_Current_Position[2] = #Destination_Station.Column) AND
                   ("Pallets_Stations".Pallets[#i].Station_Current_Position[1] = #Destination_Station.Row) THEN
                   #FoundIndex := #i;
                   EXIT;
               END_IF;
           END_FOR;
       END_IF;

   IF #FoundIndex <> 0 THEN
           IF #Pallet_Go_StD_StS THEN
               "Pallets_Stations".Pallets[#FoundIndex].Station_Current_Position[2] := "Pallets_Stations".Pallets[#FoundIndex].Station_Current_Position[2] + 1;
           ELSIF #Pallet_Go_StS_StD THEN
               "Pallets_Stations".Pallets[#FoundIndex].Station_Current_Position[2] := "Pallets_Stations".Pallets[#FoundIndex].Station_Current_Position[2] - 1;
           END_IF;
       END_IF;
END_REGION

REGION Network 7
   RUNG wire#powerrail
      Contact( #Reset_StD_StS )
      R_Coil( #HMI_StD_StS )
   END_RUNG
   RUNG wire#powerrail
      Contact( #Reset_StS_StD )
      R_Coil( #HMI_StS_StD )
   END_RUNG
   // the same network as SCL:
   IF #Reset_StD_StS THEN #HMI_StD_StS := FALSE; END_IF;
   IF #Reset_StS_StD THEN #HMI_StS_StD := FALSE; END_IF;
END_REGION

REGION Network 8 (SCL): Centering pallet
   IF NOT #isTippler AND (NOT #Destination_Station.SensorB OR
       NOT #Destination_Station.SensorC) THEN
       #oCentering := 0;
       #CenteringStep := 0;
       IF #isCentering THEN
           #Centering_Alarm := TRUE;
           #isCentering := FALSE;
       END_IF;
   END_IF;


   IF #isCentering THEN
       IF NOT #isTippler THEN
           CASE #CenteringStep OF
               0:
                   IF #Destination_Station.SensorB AND
                       #Destination_Station.SensorC AND
                       #Destination_Station.SensorA THEN
                       #Set_Speed := #SPEED_BACK;
                       //#Jog_StS := TRUE;
                       #Jog_StD := TRUE;
                   END_IF;

                   IF  #Destination_Station.SensorB AND
                       #Destination_Station.SensorC AND
                       NOT #Destination_Station.SensorA  THEN
                       #CenteringStep := 1;
                   END_IF;

               1:
                   #Set_Speed := #SPEED_FWD;
                   //  #Jog_StS := TRUE;
                   #Jog_StD := TRUE;
                   IF #Destination_Station.SensorA THEN
                       #CenteringStep := 2;
                   END_IF;

               2:
                   #Set_Speed := 0;
                   // #Jog_StS := FALSE;
                   #Jog_StD := FALSE;
                   #oCentering := TRUE;
                   #CenteringStep := 0;
                   #isCentering := FALSE;
                   #Centering_Alarm := FALSE;
           END_CASE;

       ELSIF #isTippler THEN
           CASE #CenteringStep OF
               0:
                   IF #Start_Station.SensorB AND
                       #Start_Station.SensorC THEN
                       #Set_Speed := #SPEED_BACK;
                       //#Jog_StS := TRUE;
                       #Jog_StD := TRUE;
                   END_IF;

                   IF NOT #Start_Station.SensorA AND
                       #Start_Station.SensorB AND
                       #Start_Station.SensorC AND
                       #Start_Station.SensorD THEN
                       #CenteringStep := 1;
                   END_IF;

               1:
                   #Set_Speed := #SPEED_FWD;
                   //  #Jog_StS := TRUE;
                   #Jog_StD := TRUE;
                   IF #Start_Station.SensorA THEN
                       #CenteringStep := 2;
                   END_IF;

               2:
                   #Set_Speed := 0;
                   // #Jog_StS := FALSE;
                   #Jog_StD := FALSE;
                   #oCentering := TRUE;
                   #CenteringStep := 0;
                   #isCentering := FALSE;
                   #Centering_Alarm := FALSE;
           END_CASE;
       END_IF;
   END_IF;

   #TON_Centering(IN := #isCentering,
                  PT := T#10s);

   // Wykona się tylko raz, gdy minie 10s
   IF #TON_Centering.Q THEN
       #Centering_Alarm := TRUE;
       #isCentering := FALSE;
       #CenteringStep := 0;
       #Set_Speed := 0;
       #Jog_StD := FALSE;
       #Jog_StS := FALSE;
   END_IF;



   //#trigTimeout(CLK := #TON_Centering.Q);
END_REGION

REGION Network 9: Reverse direction
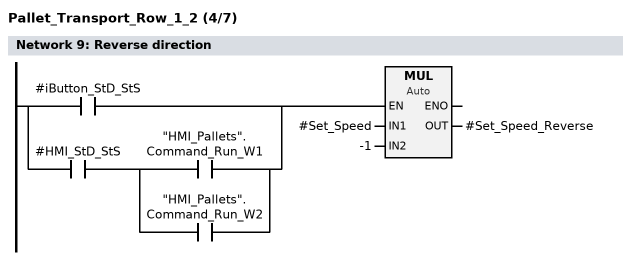
   RUNG wire#powerrail
      Contact( #iButton_StD_StS )
      wire#w1
      Mul(in1 := #Set_Speed, in2 := -1, out => #Set_Speed_Reverse)
   END_RUNG
   RUNG wire#powerrail
      Contact( #HMI_StD_StS )
      wire#w2
      Contact( "HMI_Pallets".Command_Run_W1 )
   END_RUNG wire#w1
   RUNG wire#w2
      Contact( "HMI_Pallets".Command_Run_W2 )
   END_RUNG wire#w1
   // the same network as SCL:
   IF #iButton_StD_StS OR (#HMI_StD_StS AND ("HMI_Pallets".Command_Run_W1 OR "HMI_Pallets".Command_Run_W2)) THEN
       #Set_Speed_Reverse := #Set_Speed * (-1);
   END_IF;
END_REGION

REGION Network 10: StS Drive
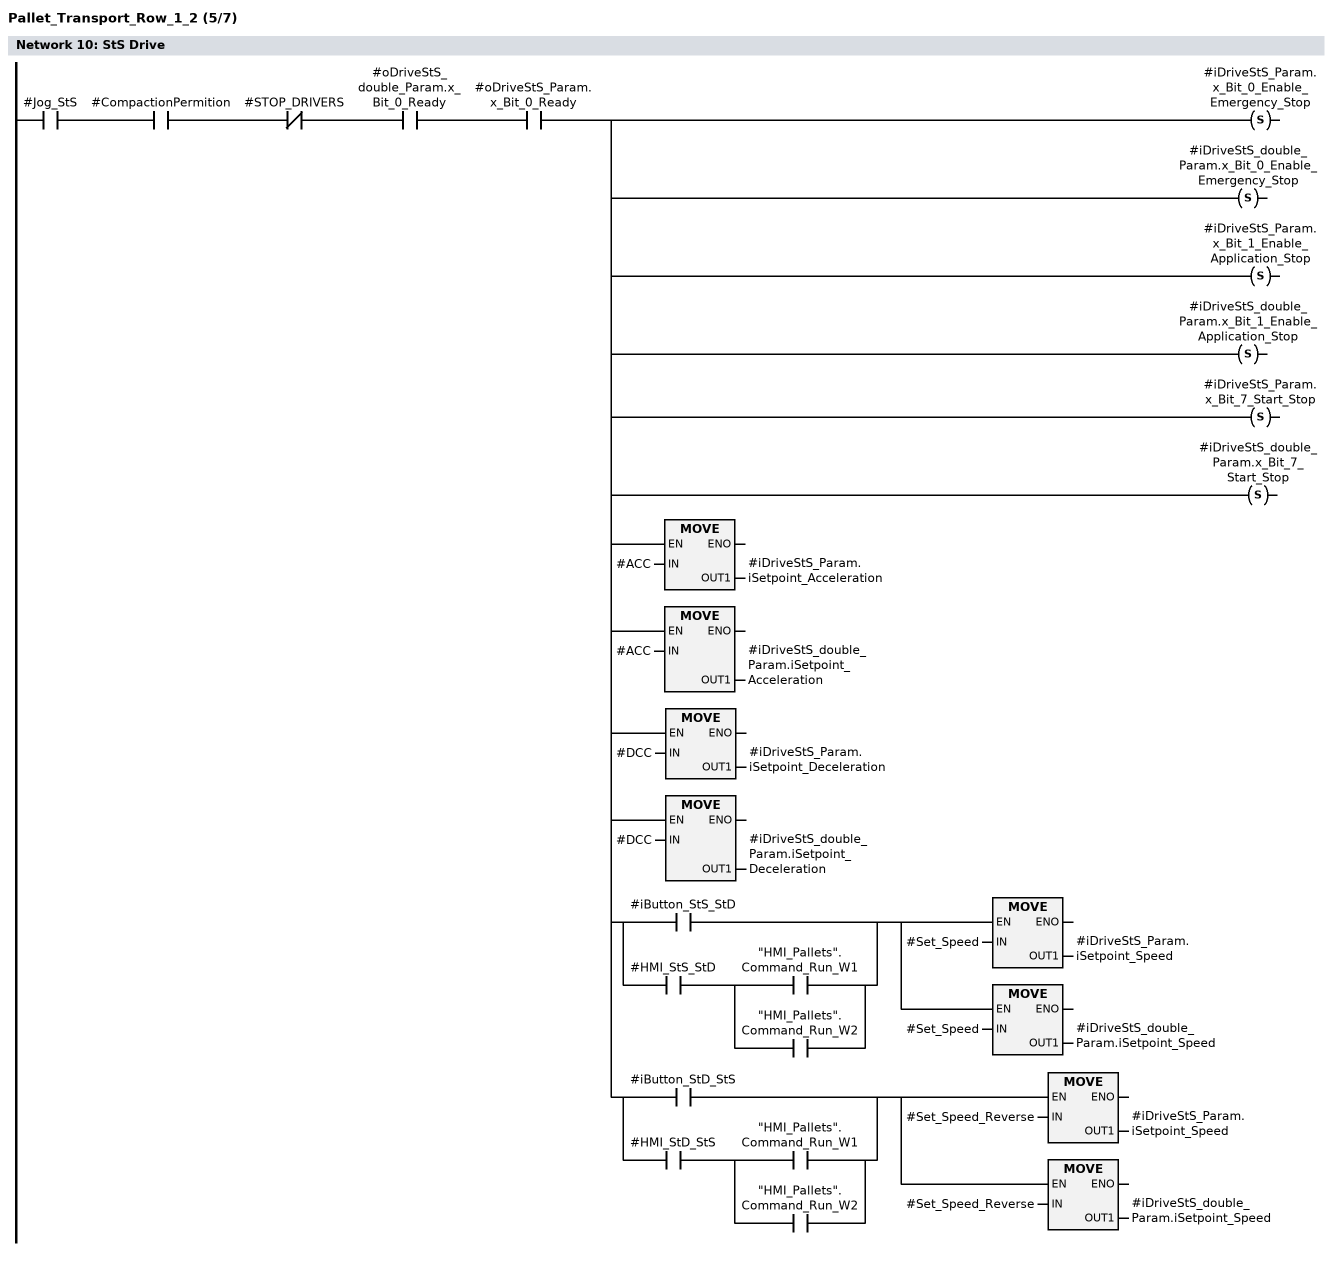
   RUNG wire#powerrail
      Contact( #Jog_StS )
      Contact( #CompactionPermition )
      I_Contact( #STOP_DRIVERS )
      Contact( #oDriveStS_double_Param.x_Bit_0_Ready )
      Contact( #oDriveStS_Param.x_Bit_0_Ready )
      wire#w1
      S_Coil( #iDriveStS_Param.x_Bit_0_Enable_Emergency_Stop )
   END_RUNG
   RUNG wire#w1
      S_Coil( #iDriveStS_double_Param.x_Bit_0_Enable_Emergency_Stop )
   END_RUNG
   RUNG wire#w1
      S_Coil( #iDriveStS_Param.x_Bit_1_Enable_Application_Stop )
   END_RUNG
   RUNG wire#w1
      S_Coil( #iDriveStS_double_Param.x_Bit_1_Enable_Application_Stop )
   END_RUNG
   RUNG wire#w1
      S_Coil( #iDriveStS_Param.x_Bit_7_Start_Stop )
   END_RUNG
   RUNG wire#w1
      S_Coil( #iDriveStS_double_Param.x_Bit_7_Start_Stop )
   END_RUNG
   RUNG wire#w1
      Move(in := #ACC, out1 => #iDriveStS_Param.iSetpoint_Acceleration)
   END_RUNG
   RUNG wire#w1
      Move(in := #ACC, out1 => #iDriveStS_double_Param.iSetpoint_Acceleration)
   END_RUNG
   RUNG wire#w1
      Move(in := #DCC, out1 => #iDriveStS_Param.iSetpoint_Deceleration)
   END_RUNG
   RUNG wire#w1
      Move(in := #DCC, out1 => #iDriveStS_double_Param.iSetpoint_Deceleration)
   END_RUNG
   RUNG wire#w1
      Contact( #iButton_StS_StD )
      wire#w2
      Move(in := #Set_Speed, out1 => #iDriveStS_Param.iSetpoint_Speed)
   END_RUNG
   RUNG wire#w1
      Contact( #HMI_StS_StD )
      wire#w3
      Contact( "HMI_Pallets".Command_Run_W1 )
   END_RUNG wire#w2
   RUNG wire#w3
      Contact( "HMI_Pallets".Command_Run_W2 )
   END_RUNG wire#w2
   RUNG wire#w2
      Move(in := #Set_Speed, out1 => #iDriveStS_double_Param.iSetpoint_Speed)
   END_RUNG
   RUNG wire#w1
      Contact( #iButton_StD_StS )
      wire#w4
      Move(in := #Set_Speed_Reverse, out1 => #iDriveStS_Param.iSetpoint_Speed)
   END_RUNG
   RUNG wire#w1
      Contact( #HMI_StD_StS )
      wire#w5
      Contact( "HMI_Pallets".Command_Run_W1 )
   END_RUNG wire#w4
   RUNG wire#w5
      Contact( "HMI_Pallets".Command_Run_W2 )
   END_RUNG wire#w4
   RUNG wire#w4
      Move(in := #Set_Speed_Reverse, out1 => #iDriveStS_double_Param.iSetpoint_Speed)
   END_RUNG
   // the same network as SCL:
   #_w1 := #Jog_StS AND #CompactionPermition AND NOT #STOP_DRIVERS AND #oDriveStS_double_Param.x_Bit_0_Ready AND #oDriveStS_Param.x_Bit_0_Ready;
   IF #_w1 THEN
       #iDriveStS_Param.x_Bit_0_Enable_Emergency_Stop := TRUE;
       #iDriveStS_double_Param.x_Bit_0_Enable_Emergency_Stop := TRUE;
       #iDriveStS_Param.x_Bit_1_Enable_Application_Stop := TRUE;
       #iDriveStS_double_Param.x_Bit_1_Enable_Application_Stop := TRUE;
       #iDriveStS_Param.x_Bit_7_Start_Stop := TRUE;
       #iDriveStS_double_Param.x_Bit_7_Start_Stop := TRUE;
       #iDriveStS_Param.iSetpoint_Acceleration := #ACC;
       #iDriveStS_double_Param.iSetpoint_Acceleration := #ACC;
       #iDriveStS_Param.iSetpoint_Deceleration := #DCC;
       #iDriveStS_double_Param.iSetpoint_Deceleration := #DCC;
   END_IF;
   IF #_w1 AND (#iButton_StS_StD OR (#HMI_StS_StD AND ("HMI_Pallets".Command_Run_W1 OR "HMI_Pallets".Command_Run_W2))) THEN
       #iDriveStS_Param.iSetpoint_Speed := #Set_Speed;
       #iDriveStS_double_Param.iSetpoint_Speed := #Set_Speed;
   END_IF;
   IF #_w1 AND (#iButton_StD_StS OR (#HMI_StD_StS AND ("HMI_Pallets".Command_Run_W1 OR "HMI_Pallets".Command_Run_W2))) THEN
       #iDriveStS_Param.iSetpoint_Speed := #Set_Speed_Reverse;
       #iDriveStS_double_Param.iSetpoint_Speed := #Set_Speed_Reverse;
   END_IF;
END_REGION

REGION Network 11: StC Drive
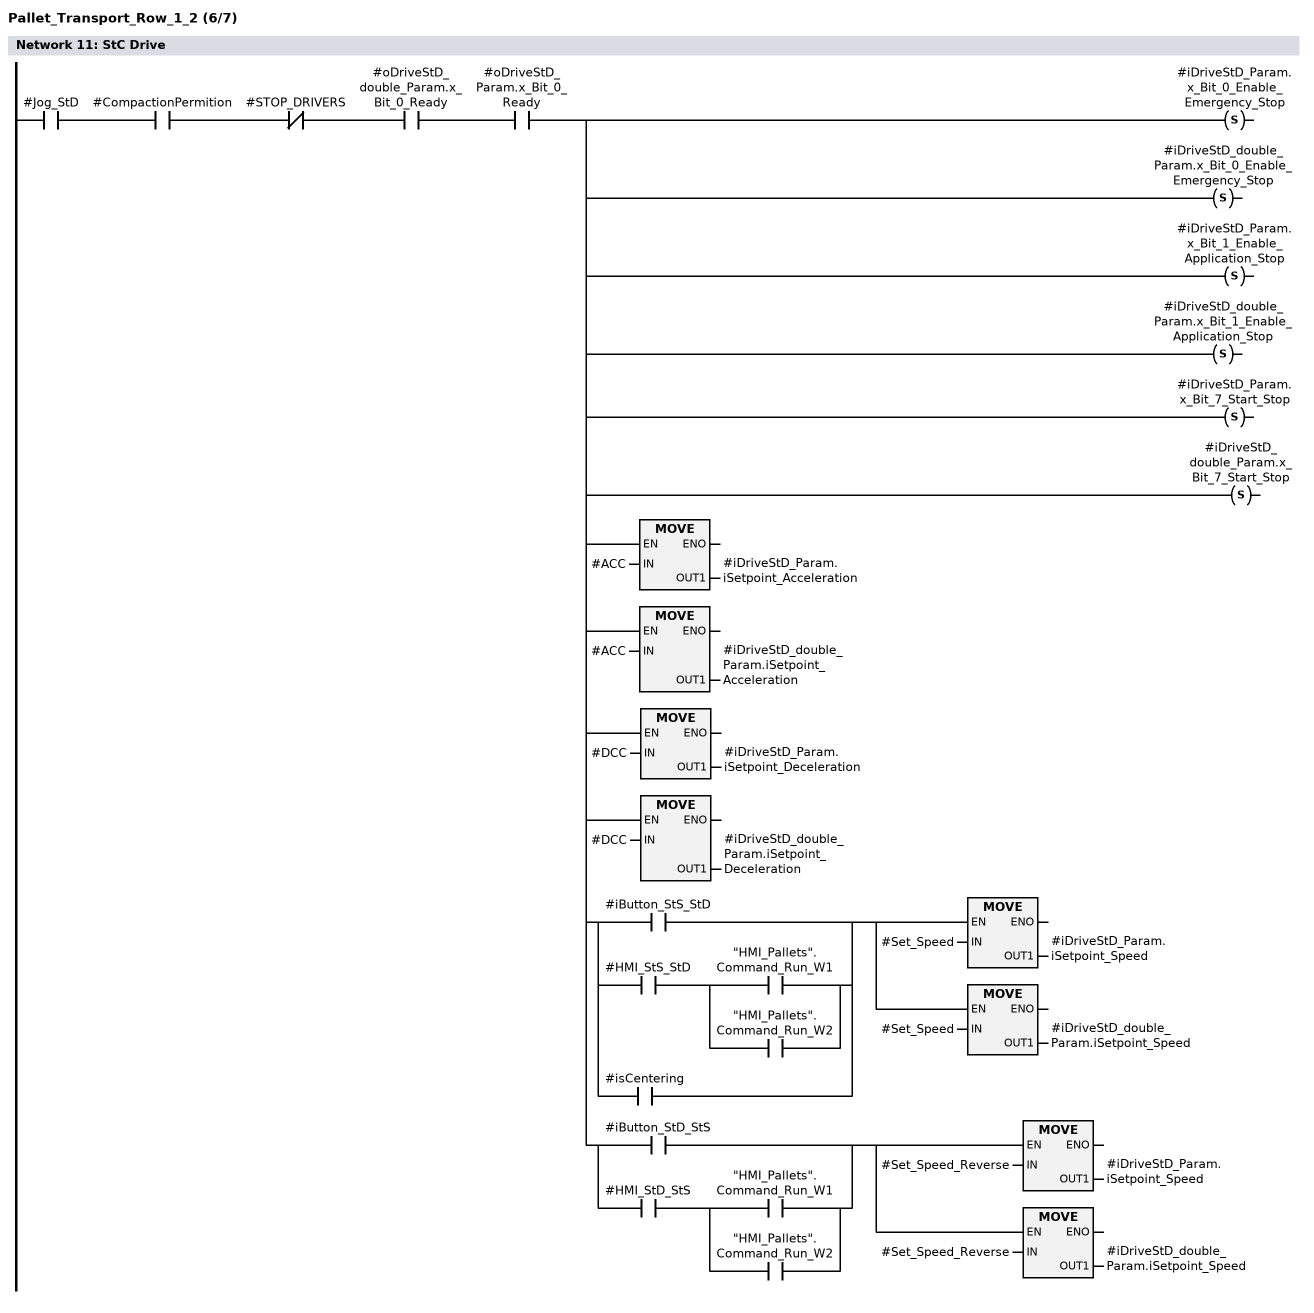
   RUNG wire#powerrail
      Contact( #Jog_StD )
      Contact( #CompactionPermition )
      I_Contact( #STOP_DRIVERS )
      Contact( #oDriveStD_double_Param.x_Bit_0_Ready )
      Contact( #oDriveStD_Param.x_Bit_0_Ready )
      wire#w1
      S_Coil( #iDriveStD_Param.x_Bit_0_Enable_Emergency_Stop )
   END_RUNG
   RUNG wire#w1
      S_Coil( #iDriveStD_double_Param.x_Bit_0_Enable_Emergency_Stop )
   END_RUNG
   RUNG wire#w1
      S_Coil( #iDriveStD_Param.x_Bit_1_Enable_Application_Stop )
   END_RUNG
   RUNG wire#w1
      S_Coil( #iDriveStD_double_Param.x_Bit_1_Enable_Application_Stop )
   END_RUNG
   RUNG wire#w1
      S_Coil( #iDriveStD_Param.x_Bit_7_Start_Stop )
   END_RUNG
   RUNG wire#w1
      S_Coil( #iDriveStD_double_Param.x_Bit_7_Start_Stop )
   END_RUNG
   RUNG wire#w1
      Move(in := #ACC, out1 => #iDriveStD_Param.iSetpoint_Acceleration)
   END_RUNG
   RUNG wire#w1
      Move(in := #ACC, out1 => #iDriveStD_double_Param.iSetpoint_Acceleration)
   END_RUNG
   RUNG wire#w1
      Move(in := #DCC, out1 => #iDriveStD_Param.iSetpoint_Deceleration)
   END_RUNG
   RUNG wire#w1
      Move(in := #DCC, out1 => #iDriveStD_double_Param.iSetpoint_Deceleration)
   END_RUNG
   RUNG wire#w1
      Contact( #iButton_StS_StD )
      wire#w2
      Move(in := #Set_Speed, out1 => #iDriveStD_Param.iSetpoint_Speed)
   END_RUNG
   RUNG wire#w1
      Contact( #HMI_StS_StD )
      wire#w3
      Contact( "HMI_Pallets".Command_Run_W1 )
   END_RUNG wire#w2
   RUNG wire#w3
      Contact( "HMI_Pallets".Command_Run_W2 )
   END_RUNG wire#w2
   RUNG wire#w1
      Contact( #isCentering )
   END_RUNG wire#w2
   RUNG wire#w2
      Move(in := #Set_Speed, out1 => #iDriveStD_double_Param.iSetpoint_Speed)
   END_RUNG
   RUNG wire#w1
      Contact( #iButton_StD_StS )
      wire#w4
      Move(in := #Set_Speed_Reverse, out1 => #iDriveStD_Param.iSetpoint_Speed)
   END_RUNG
   RUNG wire#w1
      Contact( #HMI_StD_StS )
      wire#w5
      Contact( "HMI_Pallets".Command_Run_W1 )
   END_RUNG wire#w4
   RUNG wire#w5
      Contact( "HMI_Pallets".Command_Run_W2 )
   END_RUNG wire#w4
   RUNG wire#w4
      Move(in := #Set_Speed_Reverse, out1 => #iDriveStD_double_Param.iSetpoint_Speed)
   END_RUNG
   // the same network as SCL:
   #_w1 := #Jog_StD AND #CompactionPermition AND NOT #STOP_DRIVERS AND #oDriveStD_double_Param.x_Bit_0_Ready AND #oDriveStD_Param.x_Bit_0_Ready;
   IF #_w1 THEN
       #iDriveStD_Param.x_Bit_0_Enable_Emergency_Stop := TRUE;
       #iDriveStD_double_Param.x_Bit_0_Enable_Emergency_Stop := TRUE;
       #iDriveStD_Param.x_Bit_1_Enable_Application_Stop := TRUE;
       #iDriveStD_double_Param.x_Bit_1_Enable_Application_Stop := TRUE;
       #iDriveStD_Param.x_Bit_7_Start_Stop := TRUE;
       #iDriveStD_double_Param.x_Bit_7_Start_Stop := TRUE;
       #iDriveStD_Param.iSetpoint_Acceleration := #ACC;
       #iDriveStD_double_Param.iSetpoint_Acceleration := #ACC;
       #iDriveStD_Param.iSetpoint_Deceleration := #DCC;
       #iDriveStD_double_Param.iSetpoint_Deceleration := #DCC;
   END_IF;
   IF #_w1 AND (#iButton_StS_StD OR (#HMI_StS_StD AND ("HMI_Pallets".Command_Run_W1 OR "HMI_Pallets".Command_Run_W2)) OR #isCentering) THEN
       #iDriveStD_Param.iSetpoint_Speed := #Set_Speed;
       #iDriveStD_double_Param.iSetpoint_Speed := #Set_Speed;
   END_IF;
   IF #_w1 AND (#iButton_StD_StS OR (#HMI_StD_StS AND ("HMI_Pallets".Command_Run_W1 OR "HMI_Pallets".Command_Run_W2))) THEN
       #iDriveStD_Param.iSetpoint_Speed := #Set_Speed_Reverse;
       #iDriveStD_double_Param.iSetpoint_Speed := #Set_Speed_Reverse;
   END_IF;
END_REGION

REGION Network 12: StS - > StD Status
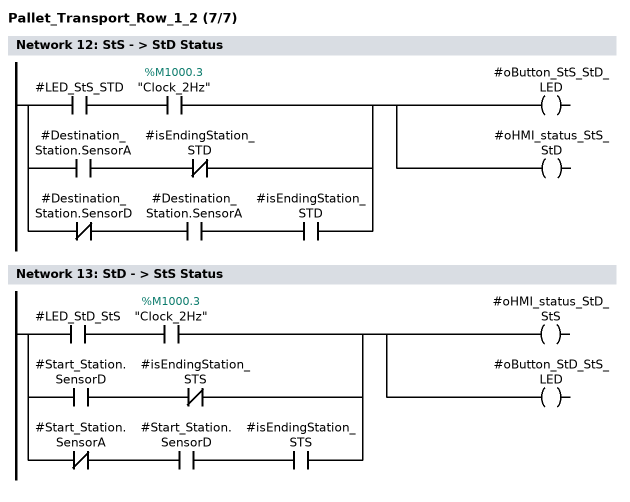
   RUNG wire#powerrail
      Contact( #LED_StS_STD )
      Contact( "Clock_2Hz" )
      wire#w1
      Coil( #oButton_StS_StD_LED )
   END_RUNG
   RUNG wire#powerrail
      Contact( #Destination_Station.SensorA )
      I_Contact( #isEndingStation_STD )
   END_RUNG wire#w1
   RUNG wire#powerrail
      I_Contact( #Destination_Station.SensorD )
      Contact( #Destination_Station.SensorA )
      Contact( #isEndingStation_STD )
   END_RUNG wire#w1
   RUNG wire#w1
      Coil( #oHMI_status_StS_StD )
   END_RUNG
   // the same network as SCL:
   #oButton_StS_StD_LED := (#LED_StS_STD AND "Clock_2Hz") OR (#Destination_Station.SensorA AND NOT #isEndingStation_STD) OR (NOT #Destination_Station.SensorD AND #Destination_Station.SensorA AND #isEndingStation_STD);
   #oHMI_status_StS_StD := #oButton_StS_StD_LED;
END_REGION

REGION Network 13: StD - > StS Status
   RUNG wire#powerrail
      Contact( #LED_StD_StS )
      Contact( "Clock_2Hz" )
      wire#w1
      Coil( #oHMI_status_StD_StS )
   END_RUNG
   RUNG wire#powerrail
      Contact( #Start_Station.SensorD )
      I_Contact( #isEndingStation_STS )
   END_RUNG wire#w1
   RUNG wire#powerrail
      I_Contact( #Start_Station.SensorA )
      Contact( #Start_Station.SensorD )
      Contact( #isEndingStation_STS )
   END_RUNG wire#w1
   RUNG wire#w1
      Coil( #oButton_StD_StS_LED )
   END_RUNG
   // the same network as SCL:
   #oHMI_status_StD_StS := (#LED_StD_StS AND "Clock_2Hz") OR (#Start_Station.SensorD AND NOT #isEndingStation_STS) OR (NOT #Start_Station.SensorA AND #Start_Station.SensorD AND #isEndingStation_STS);
   #oButton_StD_StS_LED := #oHMI_status_StD_StS;
END_REGION

REGION Network 14 (SCL): Reset centering status

   IF NOT #isTippler AND (#oCentering AND (#iDriveStD_Param.x_Bit_1_Enable_Application_Stop OR NOT #Destination_Station.SensorA)) THEN
       #oCentering := 0;
   END_IF;

   IF #isTippler AND #oCentering AND "System_To_Moving_Pallets_DB".Reset_Centering_Tippler THEN
       #oCentering := 0;
       #CenteringStep := 0;
   END_IF;
END_REGION
END_FUNCTION_BLOCK

FUNCTION_BLOCK "CentralShifter"   // FB10, LAD
{ S7_Optimized_Access := 'TRUE' }
// stored: MemoryReserve 100, SetENOAutomatically false
   VAR_INPUT
      QR_Reader : DInt;
   END_VAR
   VAR
      MC_POWER_CS_PP { S7_SetPoint := 'True'} : MC_POWER;
      MC_POWER_CS_PL { S7_SetPoint := 'True'} : MC_POWER;
      MC_POWER_CS_TP { S7_SetPoint := 'True'} : MC_POWER;
      MC_POWER_CS_TL { S7_SetPoint := 'True'} : MC_POWER;
      MC_POWER_CS_Virtual { S7_SetPoint := 'True'} : MC_POWER;
      MC_RESET_CS_PP { S7_SetPoint := 'True'} : MC_RESET;
      MC_RESET_CS_PL { S7_SetPoint := 'True'} : MC_RESET;
      MC_RESET_CS_TP { S7_SetPoint := 'True'} : MC_RESET;
      MC_RESET_CS_TL { S7_SetPoint := 'True'} : MC_RESET;
      MC_GEARIN_CS_PP { S7_SetPoint := 'True'} : MC_GEARIN;
      MC_GEARIN_CS_PL { S7_SetPoint := 'True'} : MC_GEARIN;
      MC_GEARIN_CS_TP { S7_SetPoint := 'True'} : MC_GEARIN;
      MC_GEARIN_CS_TL { S7_SetPoint := 'True'} : MC_GEARIN;
      MC_HOME_CS_PP { S7_SetPoint := 'True'} : MC_HOME;
      MC_HOME_CS_PL { S7_SetPoint := 'True'} : MC_HOME;
      MC_HOME_CS_TP { S7_SetPoint := 'True'} : MC_HOME;
      MC_HOME_CS_TL { S7_SetPoint := 'True'} : MC_HOME;
      MC_RESET_CS_Virtual { S7_SetPoint := 'True'} : MC_RESET;
      MC_MOVEJOG_CS_PL { S7_SetPoint := 'True'} : MC_MOVEJOG;
      MC_HOME_CS_Virtual { S7_SetPoint := 'True'} : MC_HOME;
      MC_MOVEJOG_CS_PP { S7_SetPoint := 'True'} : MC_MOVEJOG;
      MC_MOVEJOG_CS_TL { S7_SetPoint := 'True'} : MC_MOVEJOG;
      MC_MOVEJOG_CS_TP { S7_SetPoint := 'True'} : MC_MOVEJOG;
      MC_MOVEJOG_CS_Virtual { S7_SetPoint := 'True'} : MC_MOVEJOG;
      MC_MOVERELATIVE_CS_Virtual { S7_SetPoint := 'True'} : MC_MOVERELATIVE;
      MC_MOVEABSOLUTE_CS_Virtual { S7_SetPoint := 'True'} : MC_MOVEABSOLUTE;
      Homeing_Status { S7_SetPoint := 'True'} : Int;
      Jog_Backward_Home : Bool;
      Jog_Forward_Home : Bool;
      Jog_Velocity : Int;
      CentralShifter_Auto_Instance { S7_SetPoint := 'True'} : "CentralShifter_AutoDrive";
      Jog_Speed { S7_SetPoint := 'True'} : Real := 500.0;
      Auto_Forward : Bool;
      Auto_Backward : Bool;
      Auto_Turn_OFF { S7_SetPoint := 'True'} : TON_TIME;
      CentralShifter_SideShifters_Instance { S7_SetPoint := 'True'} : "CentralShifter_SideShifters";
      Position_To_Side_Drive { S7_SetPoint := 'True'} : Bool;
      Deceleration : Real;
      Arrived_Pos : Int;
      CS_Velocity { S7_SetPoint := 'True'} : MC_MOVEVELOCITY;
      CentralShifter_Move_Pallets_Instance { S7_SetPoint := 'True'} : "CentralShifter_Move_Pallets";
      prevBusy_Jog { S7_SetPoint := 'True'} : Bool;
      MC_SETSENSOR_Instance { S7_SetPoint := 'True'} : MC_SETSENSOR;
      prevPower { S7_SetPoint := 'True'} : Bool;
      Status_Power_Synch : Bool;
      Positions_Central : Array[7..13] of DInt;
      Central_Auto_Control_Instance { S7_SetPoint := 'True'} : "Central_Auto_Control";
      tPowerCheck { S7_SetPoint := 'True'} : TON_TIME;
      SinaParaS_CS_M_PL { S7_SetPoint := 'True'} : SinaParaS;
      SinaParaS_CS_M_PP { S7_SetPoint := 'True'} : SinaParaS;
      SinaParaS_CS_M_TL { S7_SetPoint := 'True'} : SinaParaS;
      SinaParaS_CS_M_TP { S7_SetPoint := 'True'} : SinaParaS;
      Active_Alarm { S7_SetPoint := 'True'} : Byte;
      MC_GEARINVELOCITY_pp { S7_SetPoint := 'True'} : MC_GEARINVELOCITY;
      MC_GEARINVELOCITY_tl { S7_SetPoint := 'True'} : MC_GEARINVELOCITY;
      MC_GEARINVELOCITY_tp { S7_SetPoint := 'True'} : MC_GEARINVELOCITY;
      MC_GEARINVELOCITY_pl { S7_SetPoint := 'True'} : MC_GEARINVELOCITY;
      TorqueFB_TEL750_PP { S7_SetPoint := 'True'} : "TorqueFB_TEL750";
   END_VAR
   VAR_TEMP
      temp1 : LReal;
   END_VAR
   VAR CONSTANT
      Tolerance : DInt := 13;
   END_VAR
   // Positions_Central[7] := 1080;
   // Positions_Central[8] := 15480;
   // Positions_Central[9] := 29860;
   // Positions_Central[10] := 44850;
   // Positions_Central[11] := 59230;
   // Positions_Central[12] := 73610;
   // Positions_Central[13] := 88037;
BEGIN

REGION Network 1: POWER PP
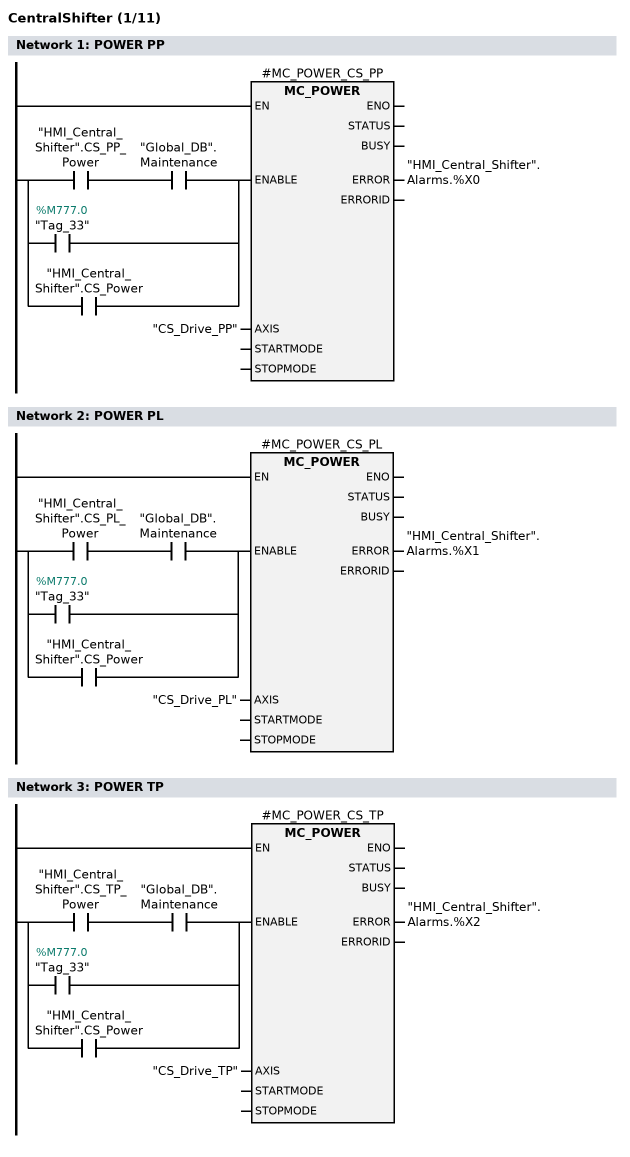
   RUNG wire#powerrail
      #MC_POWER_CS_PP.MC_POWER(Enable := wire#w1, Axis := "CS_Drive_PP", StartMode :=, StopMode :=, Status =>, Busy =>, Error => "HMI_Central_Shifter".Alarms.%X0, ErrorId =>)
   END_RUNG
   RUNG wire#powerrail
      Contact( "HMI_Central_Shifter".CS_PP_Power )
      Contact( "Global_DB".Maintenance )
   END_RUNG wire#w1
   RUNG wire#powerrail
      Contact( "Tag_33" )
   END_RUNG wire#w1
   RUNG wire#powerrail
      Contact( "HMI_Central_Shifter".CS_Power )
   END_RUNG wire#w1
   // the same network as SCL:
   #MC_POWER_CS_PP(Enable := ("HMI_Central_Shifter".CS_PP_Power AND "Global_DB".Maintenance) OR "Tag_33" OR "HMI_Central_Shifter".CS_Power,   // MC_POWER
                   Axis := "CS_Drive_PP",
                   Error => "HMI_Central_Shifter".Alarms.%X0);
END_REGION

REGION Network 2: POWER PL
   RUNG wire#powerrail
      #MC_POWER_CS_PL.MC_POWER(Enable := wire#w1, Axis := "CS_Drive_PL", StartMode :=, StopMode :=, Status =>, Busy =>, Error => "HMI_Central_Shifter".Alarms.%X1, ErrorId =>)
   END_RUNG
   RUNG wire#powerrail
      Contact( "HMI_Central_Shifter".CS_PL_Power )
      Contact( "Global_DB".Maintenance )
   END_RUNG wire#w1
   RUNG wire#powerrail
      Contact( "Tag_33" )
   END_RUNG wire#w1
   RUNG wire#powerrail
      Contact( "HMI_Central_Shifter".CS_Power )
   END_RUNG wire#w1
   // the same network as SCL:
   #MC_POWER_CS_PL(Enable := ("HMI_Central_Shifter".CS_PL_Power AND "Global_DB".Maintenance) OR "Tag_33" OR "HMI_Central_Shifter".CS_Power,   // MC_POWER
                   Axis := "CS_Drive_PL",
                   Error => "HMI_Central_Shifter".Alarms.%X1);
END_REGION

REGION Network 3: POWER TP
   RUNG wire#powerrail
      #MC_POWER_CS_TP.MC_POWER(Enable := wire#w1, Axis := "CS_Drive_TP", StartMode :=, StopMode :=, Status =>, Busy =>, Error => "HMI_Central_Shifter".Alarms.%X2, ErrorId =>)
   END_RUNG
   RUNG wire#powerrail
      Contact( "HMI_Central_Shifter".CS_TP_Power )
      Contact( "Global_DB".Maintenance )
   END_RUNG wire#w1
   RUNG wire#powerrail
      Contact( "Tag_33" )
   END_RUNG wire#w1
   RUNG wire#powerrail
      Contact( "HMI_Central_Shifter".CS_Power )
   END_RUNG wire#w1
   // the same network as SCL:
   #MC_POWER_CS_TP(Enable := ("HMI_Central_Shifter".CS_TP_Power AND "Global_DB".Maintenance) OR "Tag_33" OR "HMI_Central_Shifter".CS_Power,   // MC_POWER
                   Axis := "CS_Drive_TP",
                   Error => "HMI_Central_Shifter".Alarms.%X2);
END_REGION

REGION Network 4: POWER TL
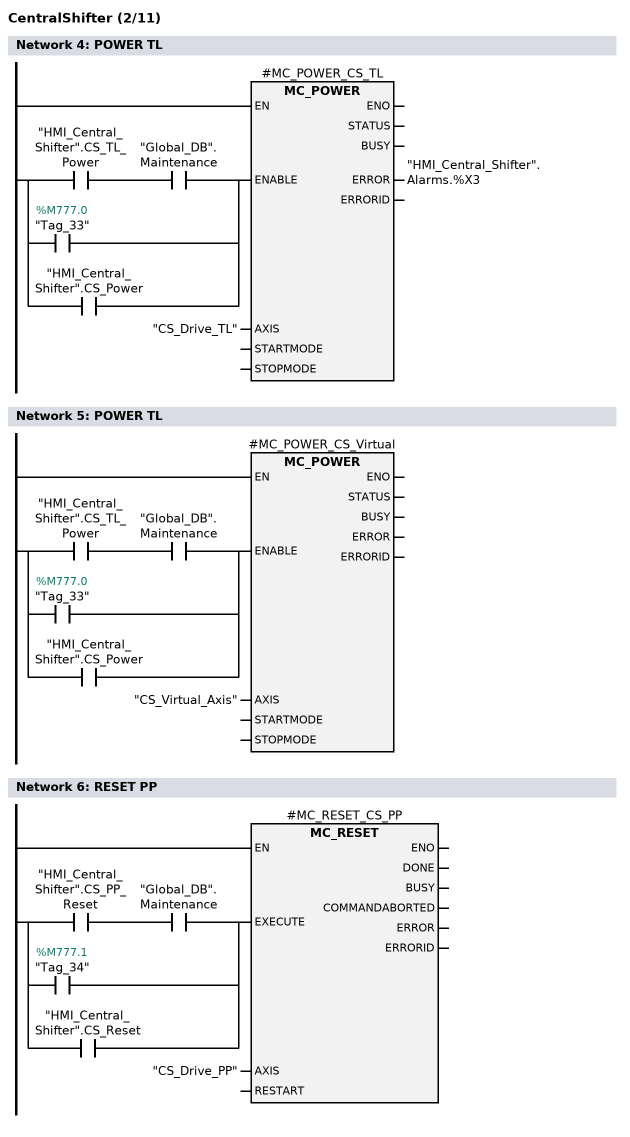
   RUNG wire#powerrail
      #MC_POWER_CS_TL.MC_POWER(Enable := wire#w1, Axis := "CS_Drive_TL", StartMode :=, StopMode :=, Status =>, Busy =>, Error => "HMI_Central_Shifter".Alarms.%X3, ErrorId =>)
   END_RUNG
   RUNG wire#powerrail
      Contact( "HMI_Central_Shifter".CS_TL_Power )
      Contact( "Global_DB".Maintenance )
   END_RUNG wire#w1
   RUNG wire#powerrail
      Contact( "Tag_33" )
   END_RUNG wire#w1
   RUNG wire#powerrail
      Contact( "HMI_Central_Shifter".CS_Power )
   END_RUNG wire#w1
   // the same network as SCL:
   #MC_POWER_CS_TL(Enable := ("HMI_Central_Shifter".CS_TL_Power AND "Global_DB".Maintenance) OR "Tag_33" OR "HMI_Central_Shifter".CS_Power,   // MC_POWER
                   Axis := "CS_Drive_TL",
                   Error => "HMI_Central_Shifter".Alarms.%X3);
END_REGION

REGION Network 5: POWER TL
   RUNG wire#powerrail
      #MC_POWER_CS_Virtual.MC_POWER(Enable := wire#w1, Axis := "CS_Virtual_Axis", StartMode :=, StopMode :=, Status =>, Busy =>, Error =>, ErrorId =>)
   END_RUNG
   RUNG wire#powerrail
      Contact( "HMI_Central_Shifter".CS_TL_Power )
      Contact( "Global_DB".Maintenance )
   END_RUNG wire#w1
   RUNG wire#powerrail
      Contact( "Tag_33" )
   END_RUNG wire#w1
   RUNG wire#powerrail
      Contact( "HMI_Central_Shifter".CS_Power )
   END_RUNG wire#w1
   // the same network as SCL:
   #MC_POWER_CS_Virtual(Enable := ("HMI_Central_Shifter".CS_TL_Power AND "Global_DB".Maintenance) OR "Tag_33" OR "HMI_Central_Shifter".CS_Power,   // MC_POWER
                        Axis := "CS_Virtual_Axis");
END_REGION

REGION Network 6: RESET PP
   RUNG wire#powerrail
      #MC_RESET_CS_PP.MC_RESET(Execute := wire#w1, Axis := "CS_Drive_PP", Restart :=, Done =>, Busy =>, CommandAborted =>, Error =>, ErrorId =>)
   END_RUNG
   RUNG wire#powerrail
      Contact( "HMI_Central_Shifter".CS_PP_Reset )
      Contact( "Global_DB".Maintenance )
   END_RUNG wire#w1
   RUNG wire#powerrail
      Contact( "Tag_34" )
   END_RUNG wire#w1
   RUNG wire#powerrail
      Contact( "HMI_Central_Shifter".CS_Reset )
   END_RUNG wire#w1
   // the same network as SCL:
   #MC_RESET_CS_PP(Execute := ("HMI_Central_Shifter".CS_PP_Reset AND "Global_DB".Maintenance) OR "Tag_34" OR "HMI_Central_Shifter".CS_Reset,   // MC_RESET
                   Axis := "CS_Drive_PP");
END_REGION

REGION Network 7: RESET PL
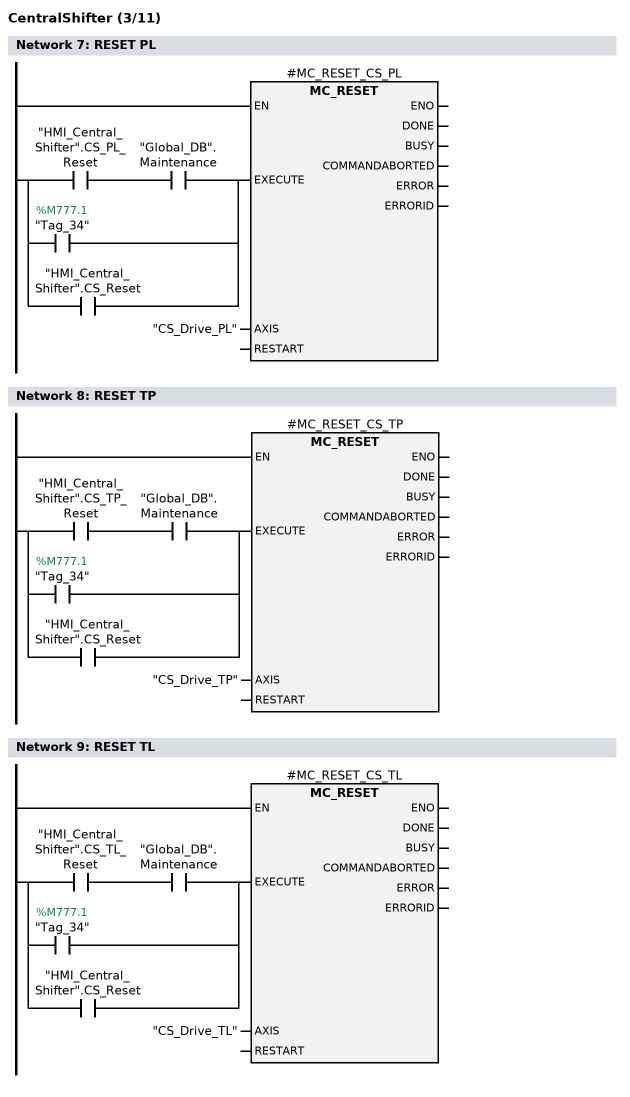
   RUNG wire#powerrail
      #MC_RESET_CS_PL.MC_RESET(Execute := wire#w1, Axis := "CS_Drive_PL", Restart :=, Done =>, Busy =>, CommandAborted =>, Error =>, ErrorId =>)
   END_RUNG
   RUNG wire#powerrail
      Contact( "HMI_Central_Shifter".CS_PL_Reset )
      Contact( "Global_DB".Maintenance )
   END_RUNG wire#w1
   RUNG wire#powerrail
      Contact( "Tag_34" )
   END_RUNG wire#w1
   RUNG wire#powerrail
      Contact( "HMI_Central_Shifter".CS_Reset )
   END_RUNG wire#w1
   // the same network as SCL:
   #MC_RESET_CS_PL(Execute := ("HMI_Central_Shifter".CS_PL_Reset AND "Global_DB".Maintenance) OR "Tag_34" OR "HMI_Central_Shifter".CS_Reset,   // MC_RESET
                   Axis := "CS_Drive_PL");
END_REGION

REGION Network 8: RESET TP
   RUNG wire#powerrail
      #MC_RESET_CS_TP.MC_RESET(Execute := wire#w1, Axis := "CS_Drive_TP", Restart :=, Done =>, Busy =>, CommandAborted =>, Error =>, ErrorId =>)
   END_RUNG
   RUNG wire#powerrail
      Contact( "HMI_Central_Shifter".CS_TP_Reset )
      Contact( "Global_DB".Maintenance )
   END_RUNG wire#w1
   RUNG wire#powerrail
      Contact( "Tag_34" )
   END_RUNG wire#w1
   RUNG wire#powerrail
      Contact( "HMI_Central_Shifter".CS_Reset )
   END_RUNG wire#w1
   // the same network as SCL:
   #MC_RESET_CS_TP(Execute := ("HMI_Central_Shifter".CS_TP_Reset AND "Global_DB".Maintenance) OR "Tag_34" OR "HMI_Central_Shifter".CS_Reset,   // MC_RESET
                   Axis := "CS_Drive_TP");
END_REGION

REGION Network 9: RESET TL
   RUNG wire#powerrail
      #MC_RESET_CS_TL.MC_RESET(Execute := wire#w1, Axis := "CS_Drive_TL", Restart :=, Done =>, Busy =>, CommandAborted =>, Error =>, ErrorId =>)
   END_RUNG
   RUNG wire#powerrail
      Contact( "HMI_Central_Shifter".CS_TL_Reset )
      Contact( "Global_DB".Maintenance )
   END_RUNG wire#w1
   RUNG wire#powerrail
      Contact( "Tag_34" )
   END_RUNG wire#w1
   RUNG wire#powerrail
      Contact( "HMI_Central_Shifter".CS_Reset )
   END_RUNG wire#w1
   // the same network as SCL:
   #MC_RESET_CS_TL(Execute := ("HMI_Central_Shifter".CS_TL_Reset AND "Global_DB".Maintenance) OR "Tag_34" OR "HMI_Central_Shifter".CS_Reset,   // MC_RESET
                   Axis := "CS_Drive_TL");
END_REGION

REGION Network 10: RESET V
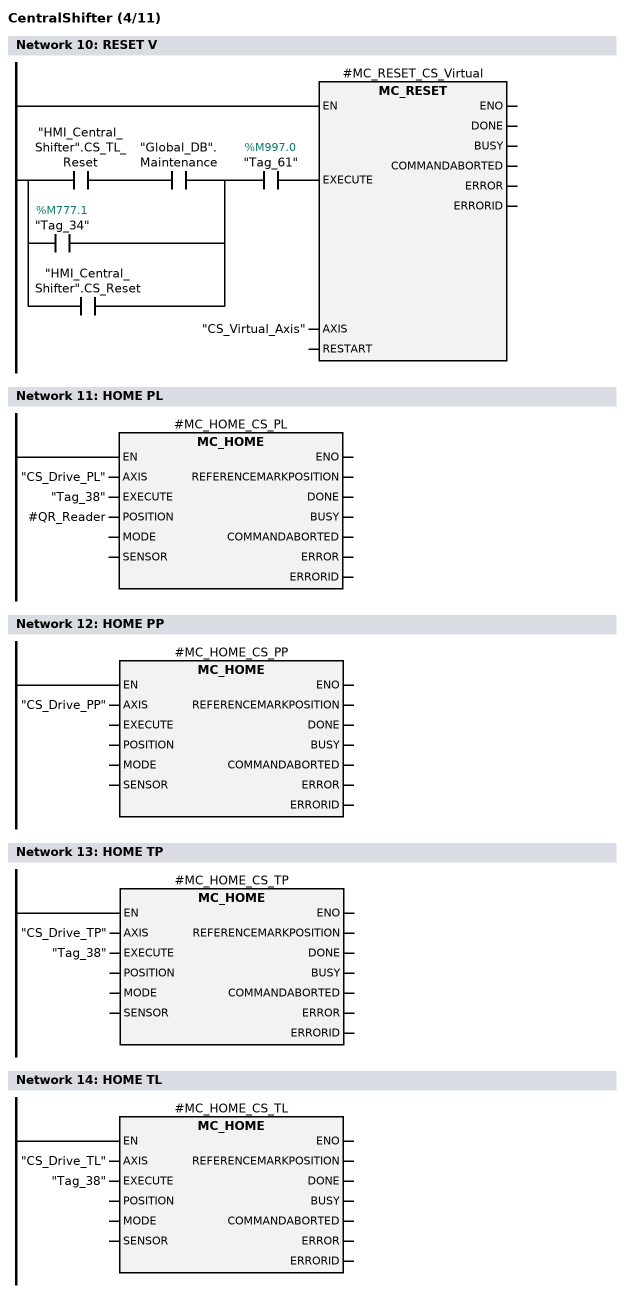
   RUNG wire#powerrail
      #MC_RESET_CS_Virtual.MC_RESET(Execute := wire#w2, Axis := "CS_Virtual_Axis", Restart :=, Done =>, Busy =>, CommandAborted =>, Error =>, ErrorId =>)
   END_RUNG
   RUNG wire#powerrail
      Contact( "HMI_Central_Shifter".CS_TL_Reset )
      Contact( "Global_DB".Maintenance )
      wire#w1
      Contact( "Tag_61" )
   END_RUNG wire#w2
   RUNG wire#powerrail
      Contact( "Tag_34" )
   END_RUNG wire#w1
   RUNG wire#powerrail
      Contact( "HMI_Central_Shifter".CS_Reset )
   END_RUNG wire#w1
   // the same network as SCL:
   #MC_RESET_CS_Virtual(Execute := (("HMI_Central_Shifter".CS_TL_Reset AND "Global_DB".Maintenance) OR "Tag_34" OR "HMI_Central_Shifter".CS_Reset) AND "Tag_61",   // MC_RESET
                        Axis := "CS_Virtual_Axis");
END_REGION

REGION Network 11: HOME PL
   RUNG wire#powerrail
      #MC_HOME_CS_PL.MC_HOME(Axis := "CS_Drive_PL", Execute := "Tag_38", Position := #QR_Reader, Mode :=, Sensor :=, ReferenceMarkPosition =>, Done =>, Busy =>, CommandAborted =>, Error =>, ErrorId =>)
   END_RUNG
   // the same network as SCL:
   #MC_HOME_CS_PL(Axis := "CS_Drive_PL", Execute := "Tag_38", Position := #QR_Reader);   // MC_HOME
END_REGION

REGION Network 12: HOME PP
   RUNG wire#powerrail
      #MC_HOME_CS_PP.MC_HOME(Axis := "CS_Drive_PP", Execute :=, Position :=, Mode :=, Sensor :=, ReferenceMarkPosition =>, Done =>, Busy =>, CommandAborted =>, Error =>, ErrorId =>)
   END_RUNG
   // the same network as SCL:
   #MC_HOME_CS_PP(Axis := "CS_Drive_PP");   // MC_HOME
END_REGION

REGION Network 13: HOME TP
   RUNG wire#powerrail
      #MC_HOME_CS_TP.MC_HOME(Axis := "CS_Drive_TP", Execute := "Tag_38", Position :=, Mode :=, Sensor :=, ReferenceMarkPosition =>, Done =>, Busy =>, CommandAborted =>, Error =>, ErrorId =>)
   END_RUNG
   // the same network as SCL:
   #MC_HOME_CS_TP(Axis := "CS_Drive_TP", Execute := "Tag_38");   // MC_HOME
END_REGION

REGION Network 14: HOME TL
   RUNG wire#powerrail
      #MC_HOME_CS_TL.MC_HOME(Axis := "CS_Drive_TL", Execute := "Tag_38", Position :=, Mode :=, Sensor :=, ReferenceMarkPosition =>, Done =>, Busy =>, CommandAborted =>, Error =>, ErrorId =>)
   END_RUNG
   // the same network as SCL:
   #MC_HOME_CS_TL(Axis := "CS_Drive_TL", Execute := "Tag_38");   // MC_HOME
END_REGION

REGION Network 15: HOME V
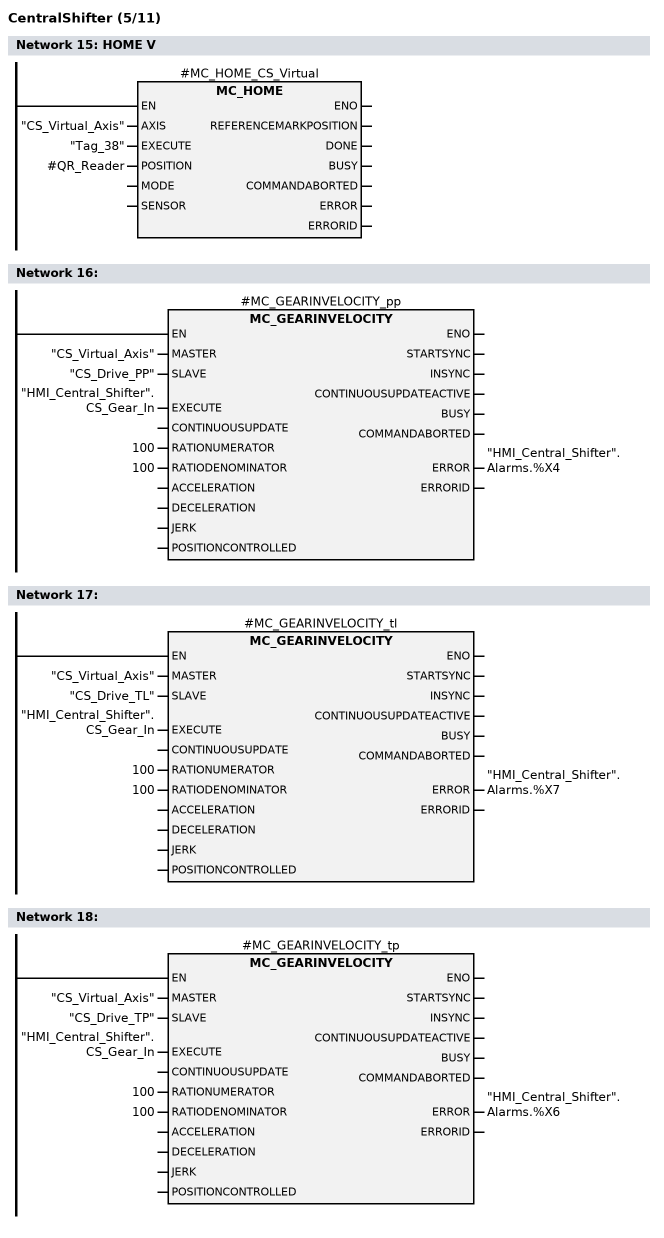
   RUNG wire#powerrail
      #MC_HOME_CS_Virtual.MC_HOME(Axis := "CS_Virtual_Axis", Execute := "Tag_38", Position := #QR_Reader, Mode :=, Sensor :=, ReferenceMarkPosition =>, Done =>, Busy =>, CommandAborted =>, Error =>, ErrorId =>)
   END_RUNG
   // the same network as SCL:
   #MC_HOME_CS_Virtual(Axis := "CS_Virtual_Axis", Execute := "Tag_38", Position := #QR_Reader);   // MC_HOME
END_REGION

REGION Network 16
   RUNG wire#powerrail
      #MC_GEARINVELOCITY_pp.MC_GEARINVELOCITY(Master := "CS_Virtual_Axis", Slave := "CS_Drive_PP", Execute := "HMI_Central_Shifter".CS_Gear_In, ContinuousUpdate :=, RatioNumerator := 100, RatioDenominator := 100, Acceleration :=, Deceleration :=, Jerk :=, PositionControlled :=, StartSync =>, InSync =>, ContinuousUpdateActive =>, Busy =>, CommandAborted =>, Error => "HMI_Central_Shifter".Alarms.%X4, ErrorId =>)
   END_RUNG
   // the same network as SCL:
   #MC_GEARINVELOCITY_pp(Master := "CS_Virtual_Axis",   // MC_GEARINVELOCITY
                         Slave := "CS_Drive_PP",
                         Execute := "HMI_Central_Shifter".CS_Gear_In,
                         RatioNumerator := 100,
                         RatioDenominator := 100,
                         Error => "HMI_Central_Shifter".Alarms.%X4);
END_REGION

REGION Network 17
   RUNG wire#powerrail
      #MC_GEARINVELOCITY_tl.MC_GEARINVELOCITY(Master := "CS_Virtual_Axis", Slave := "CS_Drive_TL", Execute := "HMI_Central_Shifter".CS_Gear_In, ContinuousUpdate :=, RatioNumerator := 100, RatioDenominator := 100, Acceleration :=, Deceleration :=, Jerk :=, PositionControlled :=, StartSync =>, InSync =>, ContinuousUpdateActive =>, Busy =>, CommandAborted =>, Error => "HMI_Central_Shifter".Alarms.%X7, ErrorId =>)
   END_RUNG
   // the same network as SCL:
   #MC_GEARINVELOCITY_tl(Master := "CS_Virtual_Axis",   // MC_GEARINVELOCITY
                         Slave := "CS_Drive_TL",
                         Execute := "HMI_Central_Shifter".CS_Gear_In,
                         RatioNumerator := 100,
                         RatioDenominator := 100,
                         Error => "HMI_Central_Shifter".Alarms.%X7);
END_REGION

REGION Network 18
   RUNG wire#powerrail
      #MC_GEARINVELOCITY_tp.MC_GEARINVELOCITY(Master := "CS_Virtual_Axis", Slave := "CS_Drive_TP", Execute := "HMI_Central_Shifter".CS_Gear_In, ContinuousUpdate :=, RatioNumerator := 100, RatioDenominator := 100, Acceleration :=, Deceleration :=, Jerk :=, PositionControlled :=, StartSync =>, InSync =>, ContinuousUpdateActive =>, Busy =>, CommandAborted =>, Error => "HMI_Central_Shifter".Alarms.%X6, ErrorId =>)
   END_RUNG
   // the same network as SCL:
   #MC_GEARINVELOCITY_tp(Master := "CS_Virtual_Axis",   // MC_GEARINVELOCITY
                         Slave := "CS_Drive_TP",
                         Execute := "HMI_Central_Shifter".CS_Gear_In,
                         RatioNumerator := 100,
                         RatioDenominator := 100,
                         Error => "HMI_Central_Shifter".Alarms.%X6);
END_REGION

REGION Network 19
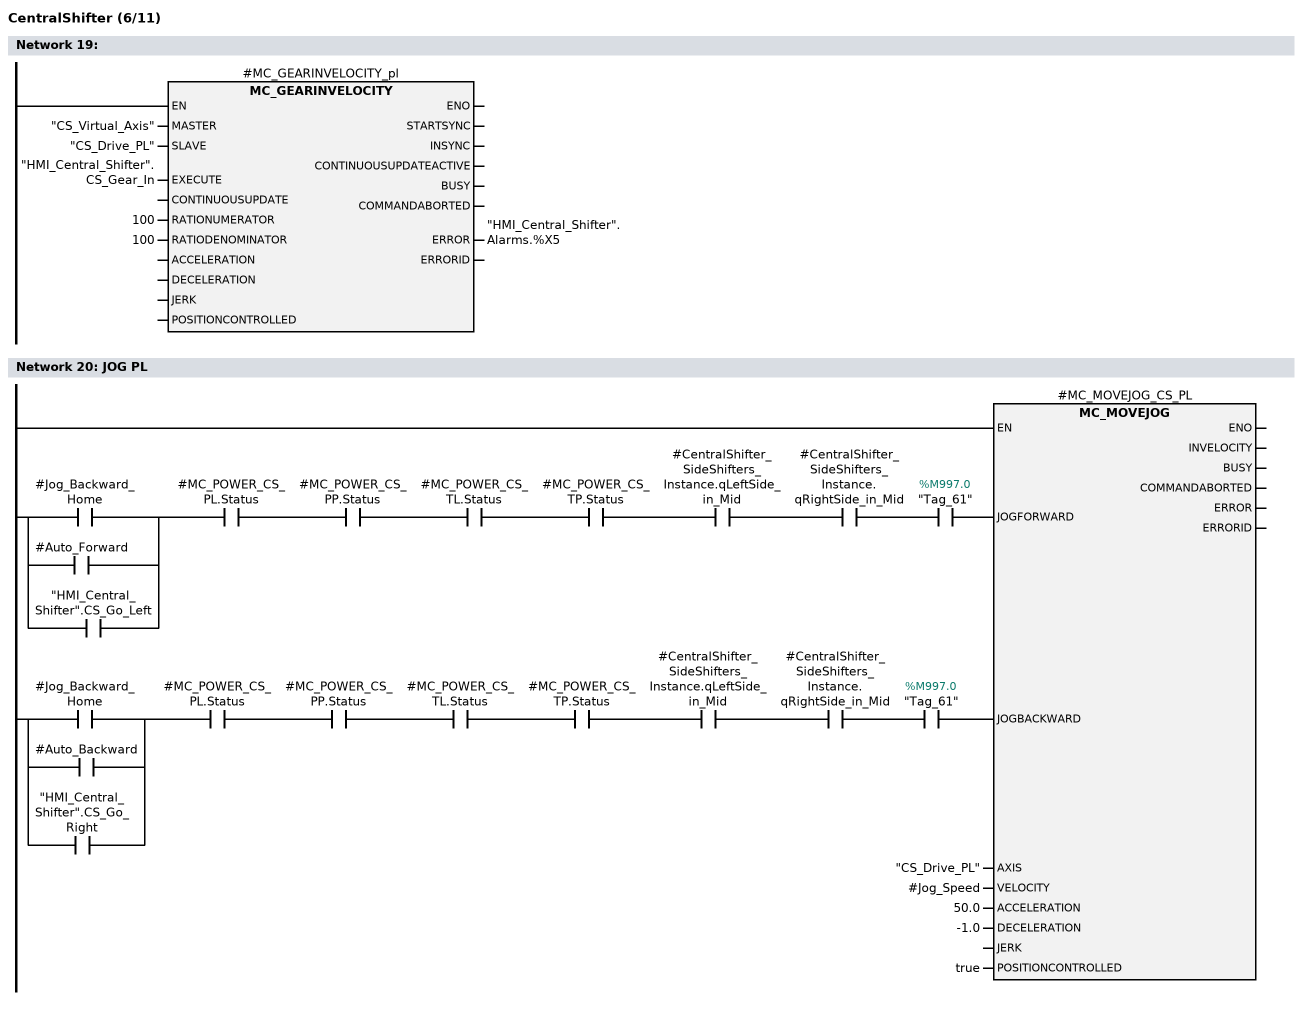
   RUNG wire#powerrail
      #MC_GEARINVELOCITY_pl.MC_GEARINVELOCITY(Master := "CS_Virtual_Axis", Slave := "CS_Drive_PL", Execute := "HMI_Central_Shifter".CS_Gear_In, ContinuousUpdate :=, RatioNumerator := 100, RatioDenominator := 100, Acceleration :=, Deceleration :=, Jerk :=, PositionControlled :=, StartSync =>, InSync =>, ContinuousUpdateActive =>, Busy =>, CommandAborted =>, Error => "HMI_Central_Shifter".Alarms.%X5, ErrorId =>)
   END_RUNG
   // the same network as SCL:
   #MC_GEARINVELOCITY_pl(Master := "CS_Virtual_Axis",   // MC_GEARINVELOCITY
                         Slave := "CS_Drive_PL",
                         Execute := "HMI_Central_Shifter".CS_Gear_In,
                         RatioNumerator := 100,
                         RatioDenominator := 100,
                         Error => "HMI_Central_Shifter".Alarms.%X5);
END_REGION

REGION Network 20: JOG PL
   RUNG wire#powerrail
      #MC_MOVEJOG_CS_PL.MC_MOVEJOG(JogForward := wire#w2, JogBackward := wire#w4, Axis := "CS_Drive_PL", Velocity := #Jog_Speed, Acceleration := 50.0, Deceleration := -1.0, Jerk :=, PositionControlled := true, InVelocity =>, Busy =>, CommandAborted =>, Error =>, ErrorId =>)
   END_RUNG
   RUNG wire#powerrail
      Contact( #Jog_Backward_Home )
      wire#w1
      Contact( #MC_POWER_CS_PL.Status )
      Contact( #MC_POWER_CS_PP.Status )
      Contact( #MC_POWER_CS_TL.Status )
      Contact( #MC_POWER_CS_TP.Status )
      Contact( #CentralShifter_SideShifters_Instance.qLeftSide_in_Mid )
      Contact( #CentralShifter_SideShifters_Instance.qRightSide_in_Mid )
      Contact( "Tag_61" )
   END_RUNG wire#w2
   RUNG wire#powerrail
      Contact( #Auto_Forward )
   END_RUNG wire#w1
   RUNG wire#powerrail
      Contact( "HMI_Central_Shifter".CS_Go_Left )
   END_RUNG wire#w1
   RUNG wire#powerrail
      Contact( #Jog_Backward_Home )
      wire#w3
      Contact( #MC_POWER_CS_PL.Status )
      Contact( #MC_POWER_CS_PP.Status )
      Contact( #MC_POWER_CS_TL.Status )
      Contact( #MC_POWER_CS_TP.Status )
      Contact( #CentralShifter_SideShifters_Instance.qLeftSide_in_Mid )
      Contact( #CentralShifter_SideShifters_Instance.qRightSide_in_Mid )
      Contact( "Tag_61" )
   END_RUNG wire#w4
   RUNG wire#powerrail
      Contact( #Auto_Backward )
   END_RUNG wire#w3
   RUNG wire#powerrail
      Contact( "HMI_Central_Shifter".CS_Go_Right )
   END_RUNG wire#w3
   // the same network as SCL:
   #MC_MOVEJOG_CS_PL(JogForward := (#Jog_Backward_Home OR #Auto_Forward OR "HMI_Central_Shifter".CS_Go_Left) AND #MC_POWER_CS_PL.Status AND #MC_POWER_CS_PP.Status AND #MC_POWER_CS_TL.Status AND #MC_POWER_CS_TP.Status AND #CentralShifter_SideShifters_Instance.qLeftSide_in_Mid AND #CentralShifter_SideShifters_Instance.qRightSide_in_Mid AND "Tag_61",   // MC_MOVEJOG
                     JogBackward := (#Jog_Backward_Home OR #Auto_Backward OR "HMI_Central_Shifter".CS_Go_Right) AND #MC_POWER_CS_PL.Status AND #MC_POWER_CS_PP.Status AND #MC_POWER_CS_TL.Status AND #MC_POWER_CS_TP.Status AND #CentralShifter_SideShifters_Instance.qLeftSide_in_Mid AND #CentralShifter_SideShifters_Instance.qRightSide_in_Mid AND "Tag_61",
                     Axis := "CS_Drive_PL",
                     Velocity := #Jog_Speed,
                     Acceleration := 50.0,
                     Deceleration := -1.0,
                     PositionControlled := true);
END_REGION

REGION Network 21: JOG PP
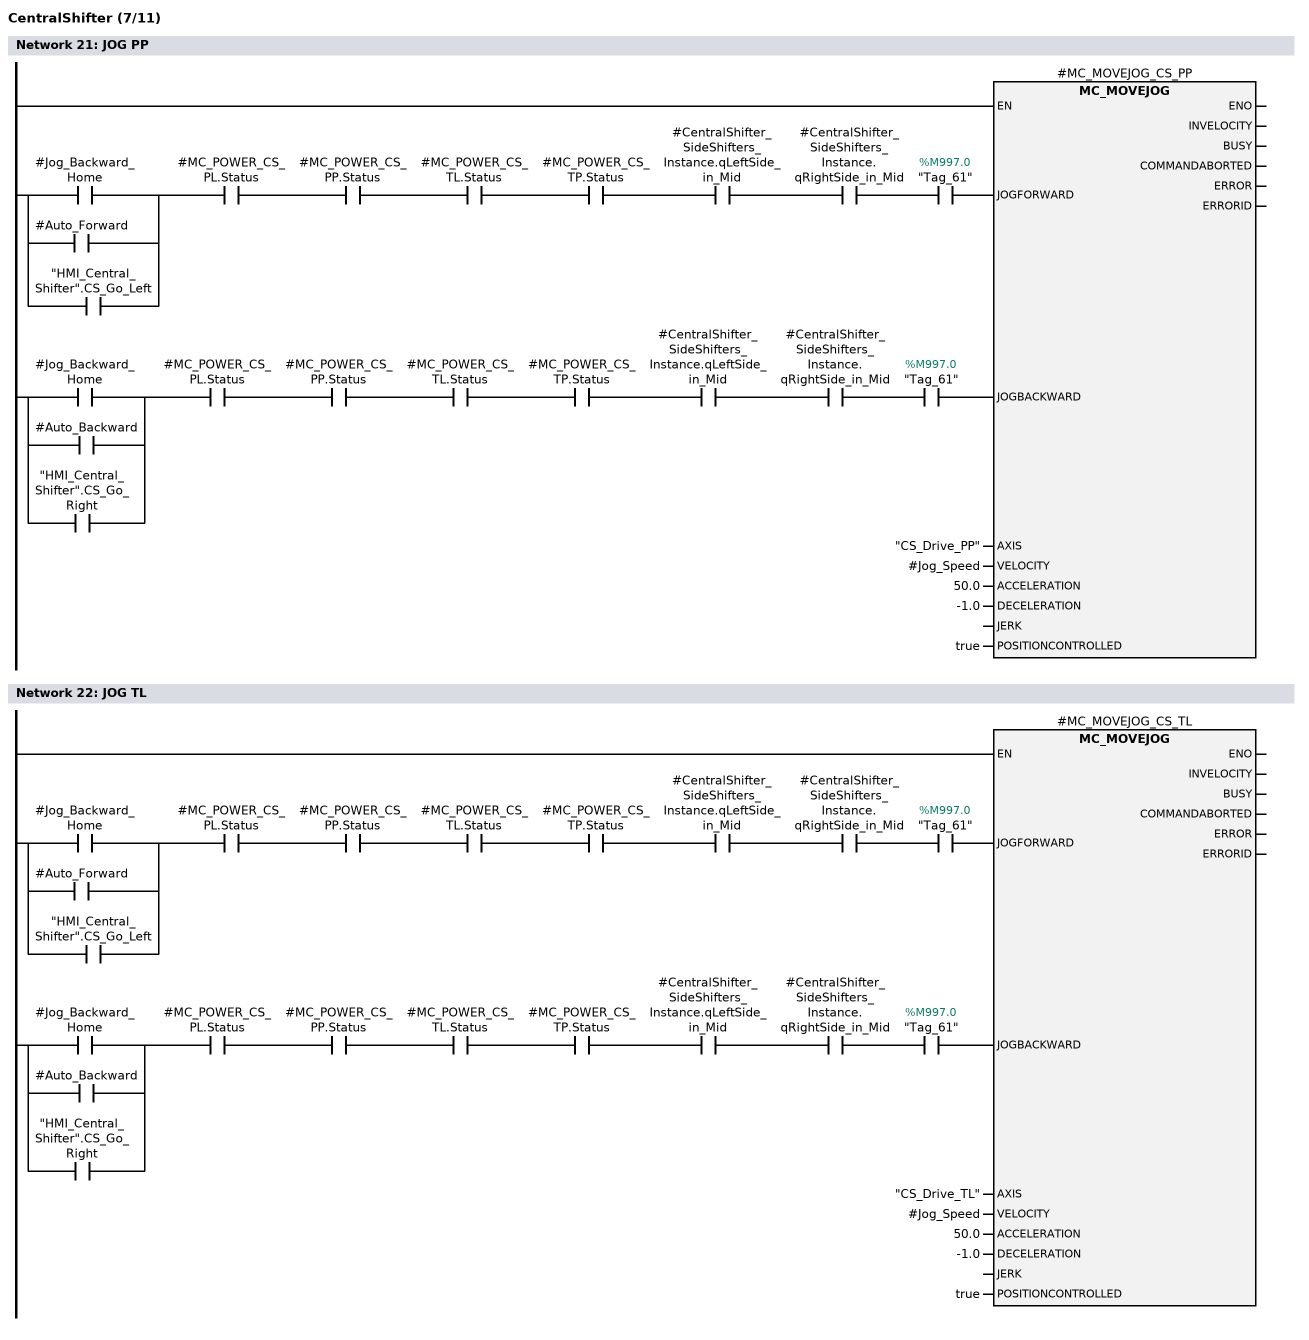
   RUNG wire#powerrail
      #MC_MOVEJOG_CS_PP.MC_MOVEJOG(JogForward := wire#w2, JogBackward := wire#w4, Axis := "CS_Drive_PP", Velocity := #Jog_Speed, Acceleration := 50.0, Deceleration := -1.0, Jerk :=, PositionControlled := true, InVelocity =>, Busy =>, CommandAborted =>, Error =>, ErrorId =>)
   END_RUNG
   RUNG wire#powerrail
      Contact( #Jog_Backward_Home )
      wire#w1
      Contact( #MC_POWER_CS_PL.Status )
      Contact( #MC_POWER_CS_PP.Status )
      Contact( #MC_POWER_CS_TL.Status )
      Contact( #MC_POWER_CS_TP.Status )
      Contact( #CentralShifter_SideShifters_Instance.qLeftSide_in_Mid )
      Contact( #CentralShifter_SideShifters_Instance.qRightSide_in_Mid )
      Contact( "Tag_61" )
   END_RUNG wire#w2
   RUNG wire#powerrail
      Contact( #Auto_Forward )
   END_RUNG wire#w1
   RUNG wire#powerrail
      Contact( "HMI_Central_Shifter".CS_Go_Left )
   END_RUNG wire#w1
   RUNG wire#powerrail
      Contact( #Jog_Backward_Home )
      wire#w3
      Contact( #MC_POWER_CS_PL.Status )
      Contact( #MC_POWER_CS_PP.Status )
      Contact( #MC_POWER_CS_TL.Status )
      Contact( #MC_POWER_CS_TP.Status )
      Contact( #CentralShifter_SideShifters_Instance.qLeftSide_in_Mid )
      Contact( #CentralShifter_SideShifters_Instance.qRightSide_in_Mid )
      Contact( "Tag_61" )
   END_RUNG wire#w4
   RUNG wire#powerrail
      Contact( #Auto_Backward )
   END_RUNG wire#w3
   RUNG wire#powerrail
      Contact( "HMI_Central_Shifter".CS_Go_Right )
   END_RUNG wire#w3
   // the same network as SCL:
   #MC_MOVEJOG_CS_PP(JogForward := (#Jog_Backward_Home OR #Auto_Forward OR "HMI_Central_Shifter".CS_Go_Left) AND #MC_POWER_CS_PL.Status AND #MC_POWER_CS_PP.Status AND #MC_POWER_CS_TL.Status AND #MC_POWER_CS_TP.Status AND #CentralShifter_SideShifters_Instance.qLeftSide_in_Mid AND #CentralShifter_SideShifters_Instance.qRightSide_in_Mid AND "Tag_61",   // MC_MOVEJOG
                     JogBackward := (#Jog_Backward_Home OR #Auto_Backward OR "HMI_Central_Shifter".CS_Go_Right) AND #MC_POWER_CS_PL.Status AND #MC_POWER_CS_PP.Status AND #MC_POWER_CS_TL.Status AND #MC_POWER_CS_TP.Status AND #CentralShifter_SideShifters_Instance.qLeftSide_in_Mid AND #CentralShifter_SideShifters_Instance.qRightSide_in_Mid AND "Tag_61",
                     Axis := "CS_Drive_PP",
                     Velocity := #Jog_Speed,
                     Acceleration := 50.0,
                     Deceleration := -1.0,
                     PositionControlled := true);
END_REGION

REGION Network 22: JOG TL
   RUNG wire#powerrail
      #MC_MOVEJOG_CS_TL.MC_MOVEJOG(JogForward := wire#w2, JogBackward := wire#w4, Axis := "CS_Drive_TL", Velocity := #Jog_Speed, Acceleration := 50.0, Deceleration := -1.0, Jerk :=, PositionControlled := true, InVelocity =>, Busy =>, CommandAborted =>, Error =>, ErrorId =>)
   END_RUNG
   RUNG wire#powerrail
      Contact( #Jog_Backward_Home )
      wire#w1
      Contact( #MC_POWER_CS_PL.Status )
      Contact( #MC_POWER_CS_PP.Status )
      Contact( #MC_POWER_CS_TL.Status )
      Contact( #MC_POWER_CS_TP.Status )
      Contact( #CentralShifter_SideShifters_Instance.qLeftSide_in_Mid )
      Contact( #CentralShifter_SideShifters_Instance.qRightSide_in_Mid )
      Contact( "Tag_61" )
   END_RUNG wire#w2
   RUNG wire#powerrail
      Contact( #Auto_Forward )
   END_RUNG wire#w1
   RUNG wire#powerrail
      Contact( "HMI_Central_Shifter".CS_Go_Left )
   END_RUNG wire#w1
   RUNG wire#powerrail
      Contact( #Jog_Backward_Home )
      wire#w3
      Contact( #MC_POWER_CS_PL.Status )
      Contact( #MC_POWER_CS_PP.Status )
      Contact( #MC_POWER_CS_TL.Status )
      Contact( #MC_POWER_CS_TP.Status )
      Contact( #CentralShifter_SideShifters_Instance.qLeftSide_in_Mid )
      Contact( #CentralShifter_SideShifters_Instance.qRightSide_in_Mid )
      Contact( "Tag_61" )
   END_RUNG wire#w4
   RUNG wire#powerrail
      Contact( #Auto_Backward )
   END_RUNG wire#w3
   RUNG wire#powerrail
      Contact( "HMI_Central_Shifter".CS_Go_Right )
   END_RUNG wire#w3
   // the same network as SCL:
   #MC_MOVEJOG_CS_TL(JogForward := (#Jog_Backward_Home OR #Auto_Forward OR "HMI_Central_Shifter".CS_Go_Left) AND #MC_POWER_CS_PL.Status AND #MC_POWER_CS_PP.Status AND #MC_POWER_CS_TL.Status AND #MC_POWER_CS_TP.Status AND #CentralShifter_SideShifters_Instance.qLeftSide_in_Mid AND #CentralShifter_SideShifters_Instance.qRightSide_in_Mid AND "Tag_61",   // MC_MOVEJOG
                     JogBackward := (#Jog_Backward_Home OR #Auto_Backward OR "HMI_Central_Shifter".CS_Go_Right) AND #MC_POWER_CS_PL.Status AND #MC_POWER_CS_PP.Status AND #MC_POWER_CS_TL.Status AND #MC_POWER_CS_TP.Status AND #CentralShifter_SideShifters_Instance.qLeftSide_in_Mid AND #CentralShifter_SideShifters_Instance.qRightSide_in_Mid AND "Tag_61",
                     Axis := "CS_Drive_TL",
                     Velocity := #Jog_Speed,
                     Acceleration := 50.0,
                     Deceleration := -1.0,
                     PositionControlled := true);
END_REGION

REGION Network 23: JOG TP
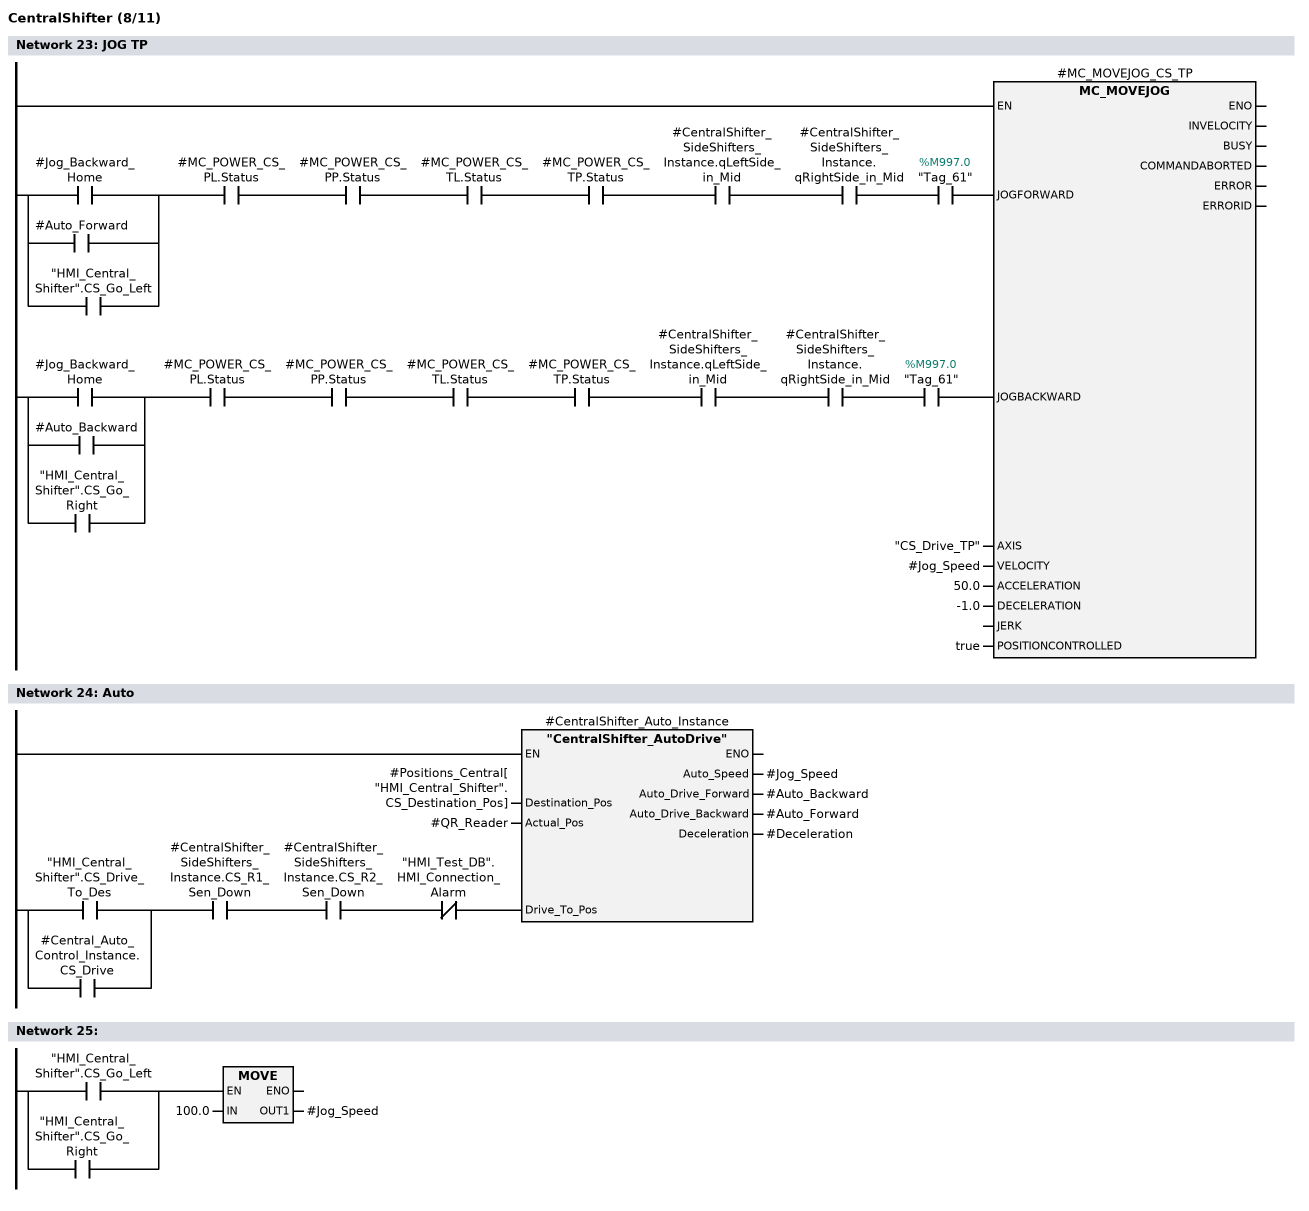
   RUNG wire#powerrail
      #MC_MOVEJOG_CS_TP.MC_MOVEJOG(JogForward := wire#w2, JogBackward := wire#w4, Axis := "CS_Drive_TP", Velocity := #Jog_Speed, Acceleration := 50.0, Deceleration := -1.0, Jerk :=, PositionControlled := true, InVelocity =>, Busy =>, CommandAborted =>, Error =>, ErrorId =>)
   END_RUNG
   RUNG wire#powerrail
      Contact( #Jog_Backward_Home )
      wire#w1
      Contact( #MC_POWER_CS_PL.Status )
      Contact( #MC_POWER_CS_PP.Status )
      Contact( #MC_POWER_CS_TL.Status )
      Contact( #MC_POWER_CS_TP.Status )
      Contact( #CentralShifter_SideShifters_Instance.qLeftSide_in_Mid )
      Contact( #CentralShifter_SideShifters_Instance.qRightSide_in_Mid )
      Contact( "Tag_61" )
   END_RUNG wire#w2
   RUNG wire#powerrail
      Contact( #Auto_Forward )
   END_RUNG wire#w1
   RUNG wire#powerrail
      Contact( "HMI_Central_Shifter".CS_Go_Left )
   END_RUNG wire#w1
   RUNG wire#powerrail
      Contact( #Jog_Backward_Home )
      wire#w3
      Contact( #MC_POWER_CS_PL.Status )
      Contact( #MC_POWER_CS_PP.Status )
      Contact( #MC_POWER_CS_TL.Status )
      Contact( #MC_POWER_CS_TP.Status )
      Contact( #CentralShifter_SideShifters_Instance.qLeftSide_in_Mid )
      Contact( #CentralShifter_SideShifters_Instance.qRightSide_in_Mid )
      Contact( "Tag_61" )
   END_RUNG wire#w4
   RUNG wire#powerrail
      Contact( #Auto_Backward )
   END_RUNG wire#w3
   RUNG wire#powerrail
      Contact( "HMI_Central_Shifter".CS_Go_Right )
   END_RUNG wire#w3
   // the same network as SCL:
   #MC_MOVEJOG_CS_TP(JogForward := (#Jog_Backward_Home OR #Auto_Forward OR "HMI_Central_Shifter".CS_Go_Left) AND #MC_POWER_CS_PL.Status AND #MC_POWER_CS_PP.Status AND #MC_POWER_CS_TL.Status AND #MC_POWER_CS_TP.Status AND #CentralShifter_SideShifters_Instance.qLeftSide_in_Mid AND #CentralShifter_SideShifters_Instance.qRightSide_in_Mid AND "Tag_61",   // MC_MOVEJOG
                     JogBackward := (#Jog_Backward_Home OR #Auto_Backward OR "HMI_Central_Shifter".CS_Go_Right) AND #MC_POWER_CS_PL.Status AND #MC_POWER_CS_PP.Status AND #MC_POWER_CS_TL.Status AND #MC_POWER_CS_TP.Status AND #CentralShifter_SideShifters_Instance.qLeftSide_in_Mid AND #CentralShifter_SideShifters_Instance.qRightSide_in_Mid AND "Tag_61",
                     Axis := "CS_Drive_TP",
                     Velocity := #Jog_Speed,
                     Acceleration := 50.0,
                     Deceleration := -1.0,
                     PositionControlled := true);
END_REGION

REGION Network 24: Auto
   RUNG wire#powerrail
      #CentralShifter_Auto_Instance(Drive_To_Pos := wire#w2, Destination_Pos := #Positions_Central["HMI_Central_Shifter".CS_Destination_Pos], Actual_Pos := #QR_Reader, Auto_Speed => #Jog_Speed, Auto_Drive_Forward => #Auto_Backward, Auto_Drive_Backward => #Auto_Forward, Deceleration => #Deceleration)
   END_RUNG
   RUNG wire#powerrail
      Contact( "HMI_Central_Shifter".CS_Drive_To_Des )
      wire#w1
      Contact( #CentralShifter_SideShifters_Instance.CS_R1_Sen_Down )
      Contact( #CentralShifter_SideShifters_Instance.CS_R2_Sen_Down )
      I_Contact( "HMI_Test_DB".HMI_Connection_Alarm )
   END_RUNG wire#w2
   RUNG wire#powerrail
      Contact( #Central_Auto_Control_Instance.CS_Drive )
   END_RUNG wire#w1
   // the same network as SCL:
   #CentralShifter_Auto_Instance(Destination_Pos := #Positions_Central["HMI_Central_Shifter".CS_Destination_Pos],   // "CentralShifter_AutoDrive"
                           Actual_Pos := #QR_Reader,
                           Drive_To_Pos := ("HMI_Central_Shifter".CS_Drive_To_Des OR #Central_Auto_Control_Instance.CS_Drive) AND #CentralShifter_SideShifters_Instance.CS_R1_Sen_Down AND #CentralShifter_SideShifters_Instance.CS_R2_Sen_Down AND NOT "HMI_Test_DB".HMI_Connection_Alarm,
                           Auto_Speed => #Jog_Speed,
                           Auto_Drive_Forward => #Auto_Backward,
                           Auto_Drive_Backward => #Auto_Forward,
                           Deceleration => #Deceleration);
END_REGION

REGION Network 25
   RUNG wire#powerrail
      Contact( "HMI_Central_Shifter".CS_Go_Left )
      wire#w1
      Move(in := 100.0, out1 => #Jog_Speed)
   END_RUNG
   RUNG wire#powerrail
      Contact( "HMI_Central_Shifter".CS_Go_Right )
   END_RUNG wire#w1
   // the same network as SCL:
   IF "HMI_Central_Shifter".CS_Go_Left OR "HMI_Central_Shifter".CS_Go_Right THEN #Jog_Speed := 100.0; END_IF;
END_REGION

REGION Network 26: JOG V
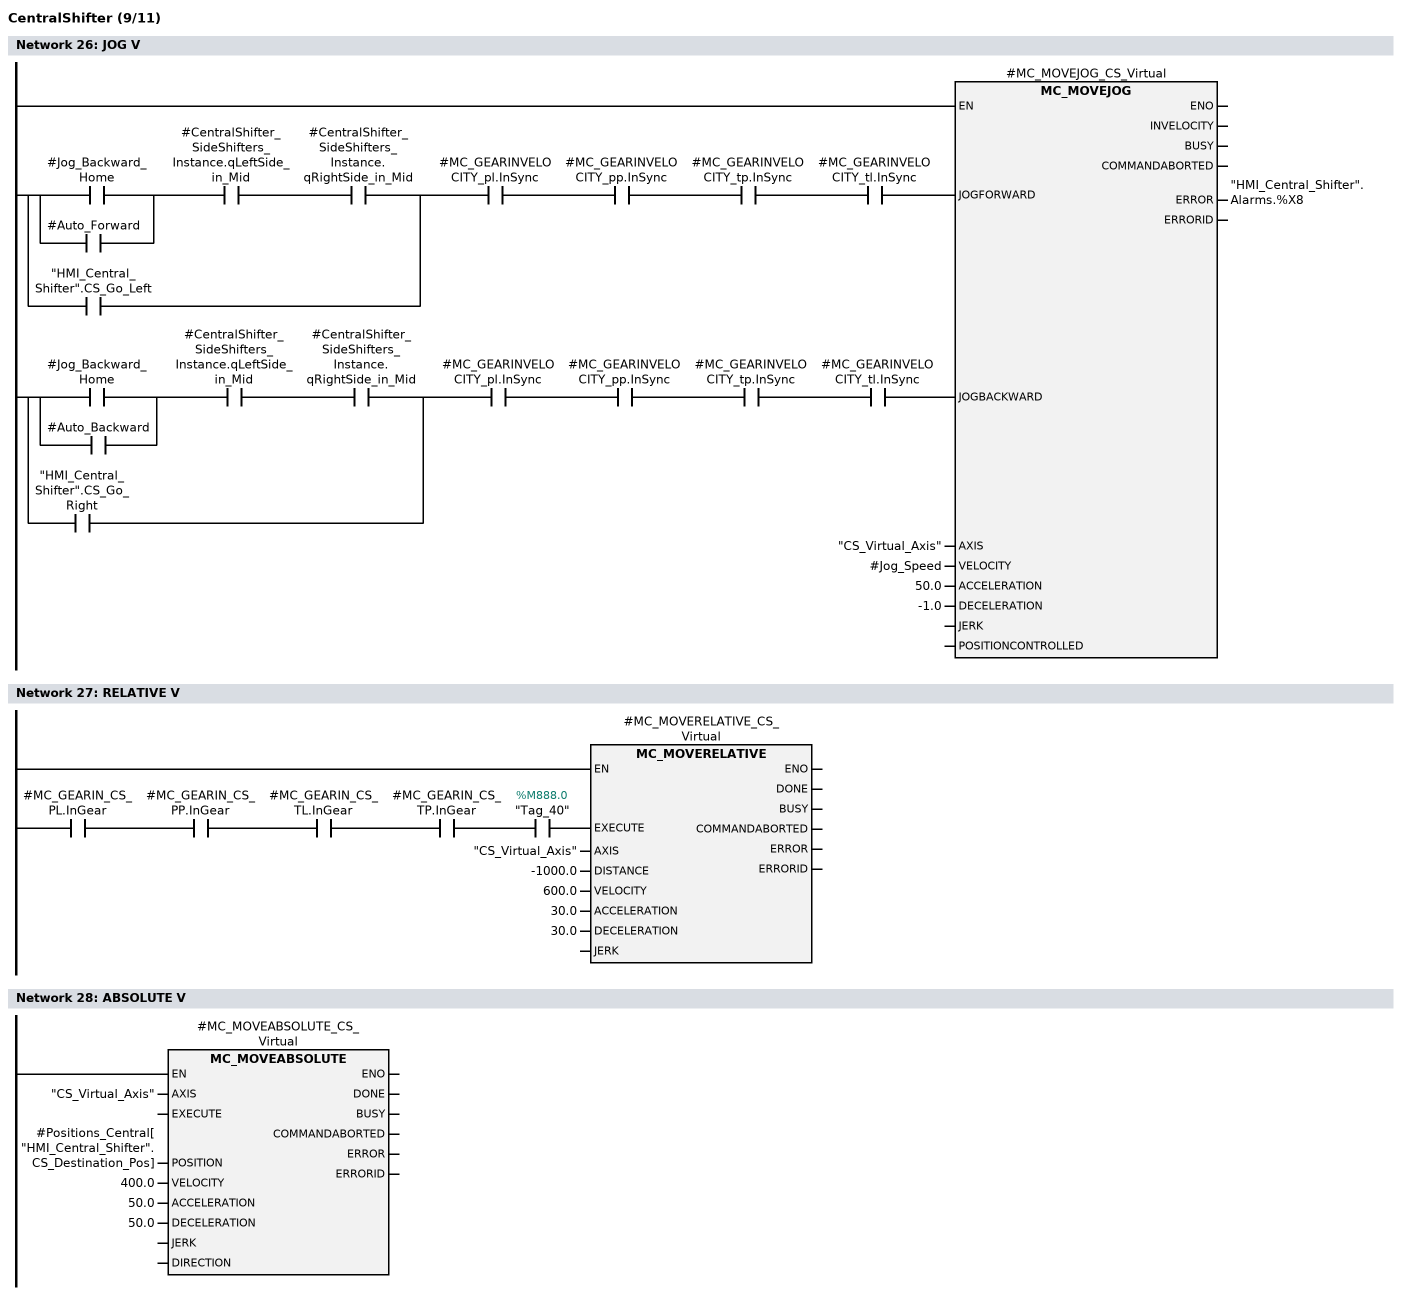
   RUNG wire#powerrail
      #MC_MOVEJOG_CS_Virtual.MC_MOVEJOG(JogForward := wire#w3, JogBackward := wire#w6, Axis := "CS_Virtual_Axis", Velocity := #Jog_Speed, Acceleration := 50.0, Deceleration := -1.0, Jerk :=, PositionControlled :=, InVelocity =>, Busy =>, CommandAborted =>, Error => "HMI_Central_Shifter".Alarms.%X8, ErrorId =>)
   END_RUNG
   RUNG wire#powerrail
      Contact( #Jog_Backward_Home )
      wire#w1
      Contact( #CentralShifter_SideShifters_Instance.qLeftSide_in_Mid )
      Contact( #CentralShifter_SideShifters_Instance.qRightSide_in_Mid )
      wire#w2
      Contact( #MC_GEARINVELOCITY_pl.InSync )
      Contact( #MC_GEARINVELOCITY_pp.InSync )
      Contact( #MC_GEARINVELOCITY_tp.InSync )
      Contact( #MC_GEARINVELOCITY_tl.InSync )
   END_RUNG wire#w3
   RUNG wire#powerrail
      Contact( #Auto_Forward )
   END_RUNG wire#w1
   RUNG wire#powerrail
      Contact( "HMI_Central_Shifter".CS_Go_Left )
   END_RUNG wire#w2
   RUNG wire#powerrail
      Contact( #Jog_Backward_Home )
      wire#w4
      Contact( #CentralShifter_SideShifters_Instance.qLeftSide_in_Mid )
      Contact( #CentralShifter_SideShifters_Instance.qRightSide_in_Mid )
      wire#w5
      Contact( #MC_GEARINVELOCITY_pl.InSync )
      Contact( #MC_GEARINVELOCITY_pp.InSync )
      Contact( #MC_GEARINVELOCITY_tp.InSync )
      Contact( #MC_GEARINVELOCITY_tl.InSync )
   END_RUNG wire#w6
   RUNG wire#powerrail
      Contact( #Auto_Backward )
   END_RUNG wire#w4
   RUNG wire#powerrail
      Contact( "HMI_Central_Shifter".CS_Go_Right )
   END_RUNG wire#w5
   // the same network as SCL:
   #MC_MOVEJOG_CS_Virtual(JogForward := (((#Jog_Backward_Home OR #Auto_Forward) AND #CentralShifter_SideShifters_Instance.qLeftSide_in_Mid AND #CentralShifter_SideShifters_Instance.qRightSide_in_Mid) OR "HMI_Central_Shifter".CS_Go_Left) AND #MC_GEARINVELOCITY_pl.InSync AND #MC_GEARINVELOCITY_pp.InSync AND #MC_GEARINVELOCITY_tp.InSync AND #MC_GEARINVELOCITY_tl.InSync,   // MC_MOVEJOG
                          JogBackward := (((#Jog_Backward_Home OR #Auto_Backward) AND #CentralShifter_SideShifters_Instance.qLeftSide_in_Mid AND #CentralShifter_SideShifters_Instance.qRightSide_in_Mid) OR "HMI_Central_Shifter".CS_Go_Right) AND #MC_GEARINVELOCITY_pl.InSync AND #MC_GEARINVELOCITY_pp.InSync AND #MC_GEARINVELOCITY_tp.InSync AND #MC_GEARINVELOCITY_tl.InSync,
                          Axis := "CS_Virtual_Axis",
                          Velocity := #Jog_Speed,
                          Acceleration := 50.0,
                          Deceleration := -1.0,
                          Error => "HMI_Central_Shifter".Alarms.%X8);
END_REGION

REGION Network 27: RELATIVE V
   RUNG wire#powerrail
      #MC_MOVERELATIVE_CS_Virtual.MC_MOVERELATIVE(Execute := wire#w1, Axis := "CS_Virtual_Axis", Distance := -1000.0, Velocity := 600.0, Acceleration := 30.0, Deceleration := 30.0, Jerk :=, Done =>, Busy =>, CommandAborted =>, Error =>, ErrorId =>)
   END_RUNG
   RUNG wire#powerrail
      Contact( #MC_GEARIN_CS_PL.InGear )
      Contact( #MC_GEARIN_CS_PP.InGear )
      Contact( #MC_GEARIN_CS_TL.InGear )
      Contact( #MC_GEARIN_CS_TP.InGear )
      Contact( "Tag_40" )
   END_RUNG wire#w1
   // the same network as SCL:
   #MC_MOVERELATIVE_CS_Virtual(Execute := #MC_GEARIN_CS_PL.InGear AND #MC_GEARIN_CS_PP.InGear AND #MC_GEARIN_CS_TL.InGear AND #MC_GEARIN_CS_TP.InGear AND "Tag_40",   // MC_MOVERELATIVE
                           Axis := "CS_Virtual_Axis",
                           Distance := -1000.0,
                           Velocity := 600.0,
                           Acceleration := 30.0,
                           Deceleration := 30.0);
END_REGION

REGION Network 28: ABSOLUTE V
   RUNG wire#powerrail
      #MC_MOVEABSOLUTE_CS_Virtual.MC_MOVEABSOLUTE(Axis := "CS_Virtual_Axis", Execute :=, Position := #Positions_Central["HMI_Central_Shifter".CS_Destination_Pos], Velocity := 400.0, Acceleration := 50.0, Deceleration := 50.0, Jerk :=, Direction :=, Done =>, Busy =>, CommandAborted =>, Error =>, ErrorId =>)
   END_RUNG
   // the same network as SCL:
   #MC_MOVEABSOLUTE_CS_Virtual(Axis := "CS_Virtual_Axis",   // MC_MOVEABSOLUTE
                           Position := #Positions_Central["HMI_Central_Shifter".CS_Destination_Pos],
                           Velocity := 400.0,
                           Acceleration := 50.0,
                           Deceleration := 50.0);
END_REGION

REGION Network 29: Auto Turn Off
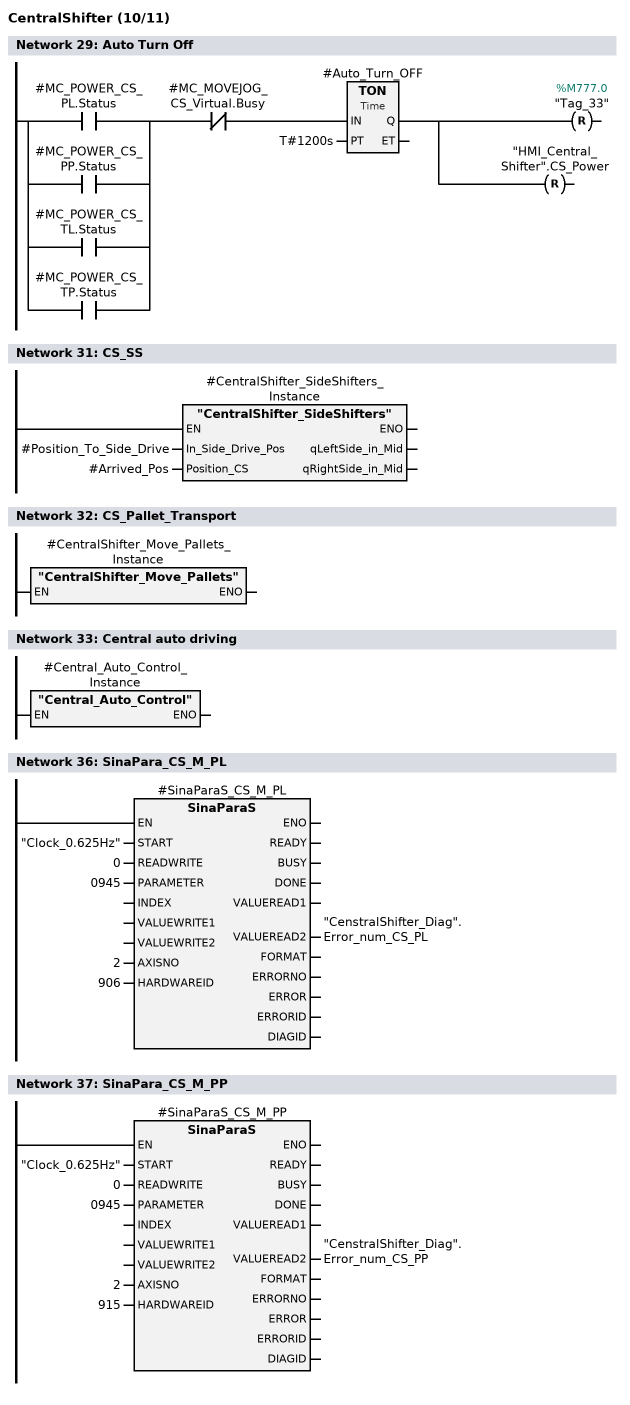
   RUNG wire#powerrail
      Contact( #MC_POWER_CS_PL.Status )
      wire#w1
      I_Contact( #MC_MOVEJOG_CS_Virtual.Busy )
      { S7_Templates := "time_type := Time" } #Auto_Turn_OFF.TON(pt := T#1200s, et =>)
      wire#w2
      R_Coil( "Tag_33" )
   END_RUNG
   RUNG wire#powerrail
      Contact( #MC_POWER_CS_PP.Status )
   END_RUNG wire#w1
   RUNG wire#powerrail
      Contact( #MC_POWER_CS_TL.Status )
   END_RUNG wire#w1
   RUNG wire#powerrail
      Contact( #MC_POWER_CS_TP.Status )
   END_RUNG wire#w1
   RUNG wire#w2
      R_Coil( "HMI_Central_Shifter".CS_Power )
   END_RUNG
   // the same network as SCL:
   #Auto_Turn_OFF(IN := (#MC_POWER_CS_PL.Status OR #MC_POWER_CS_PP.Status OR #MC_POWER_CS_TL.Status OR #MC_POWER_CS_TP.Status) AND NOT #MC_MOVEJOG_CS_Virtual.Busy,   // TON
                  PT := T#1200s);
   IF #Auto_Turn_OFF.Q THEN
       "Tag_33" := FALSE;
       "HMI_Central_Shifter".CS_Power := FALSE;
   END_IF;
END_REGION

REGION Network 30 (SCL): Position To Side Shifters Drive
   #Arrived_Pos := 0; // Reset pozycji na początku

   IF ABS(#QR_Reader - #Positions_Central[7]) <= #Tolerance THEN
       #Arrived_Pos := 7;
   ELSIF ABS(#QR_Reader - #Positions_Central[8]) <= #Tolerance THEN
       #Arrived_Pos := 8;
   ELSIF ABS(#QR_Reader - #Positions_Central[9]) <= #Tolerance THEN
       #Arrived_Pos := 9;
   ELSIF ABS(#QR_Reader - #Positions_Central[10]) <= #Tolerance THEN
       #Arrived_Pos := 10;
   ELSIF ABS(#QR_Reader - #Positions_Central[11]) <= #Tolerance THEN
       #Arrived_Pos := 11;
   ELSIF ABS(#QR_Reader - #Positions_Central[12]) <= #Tolerance THEN
       #Arrived_Pos := 12;
   ELSIF ABS(#QR_Reader - #Positions_Central[13]) <= #Tolerance THEN
       #Arrived_Pos := 13;
   END_IF;

   // Ustawienie Position_To_Side_Drive tylko jeśli coś wykryto
   IF #Arrived_Pos <> 0 THEN
       #Position_To_Side_Drive := 1;
   ELSE
       #Position_To_Side_Drive := 0;
   END_IF;
END_REGION

REGION Network 31: CS_SS
   RUNG wire#powerrail
      #CentralShifter_SideShifters_Instance(In_Side_Drive_Pos := #Position_To_Side_Drive, Position_CS := #Arrived_Pos, qLeftSide_in_Mid =>, qRightSide_in_Mid =>)
   END_RUNG
   // the same network as SCL:
   #CentralShifter_SideShifters_Instance(In_Side_Drive_Pos := #Position_To_Side_Drive,   // "CentralShifter_SideShifters"
                           Position_CS := #Arrived_Pos);
END_REGION

REGION Network 32: CS_Pallet_Transport
   RUNG wire#powerrail
      #CentralShifter_Move_Pallets_Instance()
   END_RUNG
   // the same network as SCL:
   #CentralShifter_Move_Pallets_Instance();   // "CentralShifter_Move_Pallets"
END_REGION

REGION Network 33: Central auto driving
   RUNG wire#powerrail
      #Central_Auto_Control_Instance()
   END_RUNG
   // the same network as SCL:
   #Central_Auto_Control_Instance();   // "Central_Auto_Control"
END_REGION

REGION Network 34 (SCL): Auto centering pallet
   IF (NOT #MC_MOVEJOG_CS_Virtual.Busy AND #prevBusy_Jog) OR (#MC_MOVEJOG_CS_Virtual.Busy AND NOT #prevBusy_Jog) THEN
       "HMI_Central_Shifter".CS_Pallet_Centering := TRUE;
   END_IF;

   #prevBusy_Jog:= #MC_MOVEJOG_CS_Virtual.Busy;
END_REGION

REGION Network 35 (SCL): Power - Resert - Synch HMI
   // --- Central Shifter Power Logic z opóźnieniem sprawdzania statusów ---
   (*
   // Zbocze narastające Power
   IF "HMI_Central_Shifter".CS_Power AND NOT #prevPower THEN
       "HMI_Central_Shifter".CS_Reset := TRUE;
       #tPowerCheck(IN := TRUE,
                    PT := T#2S);   // uruchom 2-sekundowy timer

   ELSIF "HMI_Central_Shifter".CS_Power AND "HMI_Central_Shifter".CS_Reset THEN
       // Po jednym cyklu reset wyłącz
       "HMI_Central_Shifter".CS_Reset := FALSE;
   END_IF;

   // Aktualizacja timera (musi być poza IF, żeby działał ciągle)
   #tPowerCheck.IN := "HMI_Central_Shifter".CS_Power;

   // Główna logika sprawdzania statusów
   IF "HMI_Central_Shifter".CS_Power AND #tPowerCheck.Q THEN
       // Sprawdź statusy dopiero po upływie czasu (gdy napędy zdążą się uruchomić)
       IF NOT (
           #MC_POWER_CS_PL.Status AND
           #MC_POWER_CS_PP.Status AND
           #MC_POWER_CS_TL.Status AND
           #MC_POWER_CS_TP.Status
           ) THEN
           // Gdy któryś napęd nie ma Power po czasie → wyłącz
           "HMI_Central_Shifter".CS_Power := FALSE;
       END_IF;

   ELSIF NOT "HMI_Central_Shifter".CS_Power THEN
       // Power OFF → reset timera i czyszczenie
       "HMI_Central_Shifter".CS_Reset := FALSE;
       #tPowerCheck.IN := FALSE;
   END_IF;

   IF #MC_POWER_CS_PP.Status AND
       #MC_POWER_CS_TL.Status AND
       #MC_POWER_CS_TP.Status THEN
       #Status_Power_Synch := 1;
   ELSE
       #Status_Power_Synch := 0;
   END_IF;

   // Zapamiętaj poprzedni stan Power
   #prevPower := "HMI_Central_Shifter".CS_Power;
   *)
   IF "HMI_Central_Shifter".CS_Sides_Go_Up OR "HMI_Central_Shifter".CS_Sides_Go_Mid OR "HMI_Central_Shifter".CS_Sides_Go_Down THEN
       "HMI_Central_Shifter".CS_Power := 0;
   END_IF;

   IF "HMI_Central_Shifter".CS_Power AND NOT #prevPower THEN
       "HMI_Central_Shifter".CS_Reset := 1;

   ELSIF "HMI_Central_Shifter".CS_Power 
         AND "HMI_Central_Shifter".CS_Reset THEN
       "HMI_Central_Shifter".CS_Reset := 0;

   ELSIF "HMI_Central_Shifter".CS_Power
         AND #MC_POWER_CS_PL.Status
         AND #MC_POWER_CS_PP.Status
         AND #MC_POWER_CS_TL.Status
         AND #MC_POWER_CS_TP.Status THEN
       "HMI_Central_Shifter".CS_Gear_In := 1;

   ELSIF "HMI_Central_Shifter".CS_Power
         AND (NOT #MC_GEARIN_CS_PL.InGear
              OR NOT #MC_GEARIN_CS_PP.InGear
              OR NOT #MC_GEARIN_CS_TP.InGear
              OR NOT #MC_GEARIN_CS_TL.InGear)
         AND NOT "HMI_Central_Shifter".CS_Reset
         AND "HMI_Central_Shifter".CS_Gear_In THEN
       "HMI_Central_Shifter".CS_Power := 0;

   ELSIF NOT "HMI_Central_Shifter".CS_Power THEN
       "HMI_Central_Shifter".CS_Reset := 0;
       "HMI_Central_Shifter".CS_Gear_In := 0;
   END_IF;

   #prevPower := "HMI_Central_Shifter".CS_Power;
END_REGION

REGION Network 36: SinaPara_CS_M_PL
   RUNG wire#powerrail
      #SinaParaS_CS_M_PL.SinaParaS(Start := "Clock_0.625Hz", ReadWrite := 0, Parameter := 0945, Index :=, ValueWrite1 :=, ValueWrite2 :=, AxisNo := 2, hardwareId := 906, Ready =>, Busy =>, Done =>, ValueRead1 =>, ValueRead2 => "CenstralShifter_Diag".Error_num_CS_PL, Format =>, ErrorNo =>, Error =>, ErrorId =>, DiagId =>)
   END_RUNG
   // the same network as SCL:
   #SinaParaS_CS_M_PL(Start := "Clock_0.625Hz",   // SinaParaS
                      ReadWrite := 0,
                      Parameter := 0945,
                      AxisNo := 2,
                      hardwareId := 906,
                      ValueRead2 => "CenstralShifter_Diag".Error_num_CS_PL);
END_REGION

REGION Network 37: SinaPara_CS_M_PP
   RUNG wire#powerrail
      #SinaParaS_CS_M_PP.SinaParaS(Start := "Clock_0.625Hz", ReadWrite := 0, Parameter := 0945, Index :=, ValueWrite1 :=, ValueWrite2 :=, AxisNo := 2, hardwareId := 915, Ready =>, Busy =>, Done =>, ValueRead1 =>, ValueRead2 => "CenstralShifter_Diag".Error_num_CS_PP, Format =>, ErrorNo =>, Error =>, ErrorId =>, DiagId =>)
   END_RUNG
   // the same network as SCL:
   #SinaParaS_CS_M_PP(Start := "Clock_0.625Hz",   // SinaParaS
                      ReadWrite := 0,
                      Parameter := 0945,
                      AxisNo := 2,
                      hardwareId := 915,
                      ValueRead2 => "CenstralShifter_Diag".Error_num_CS_PP);
END_REGION

REGION Network 38: SinaPara_CS_M_TL
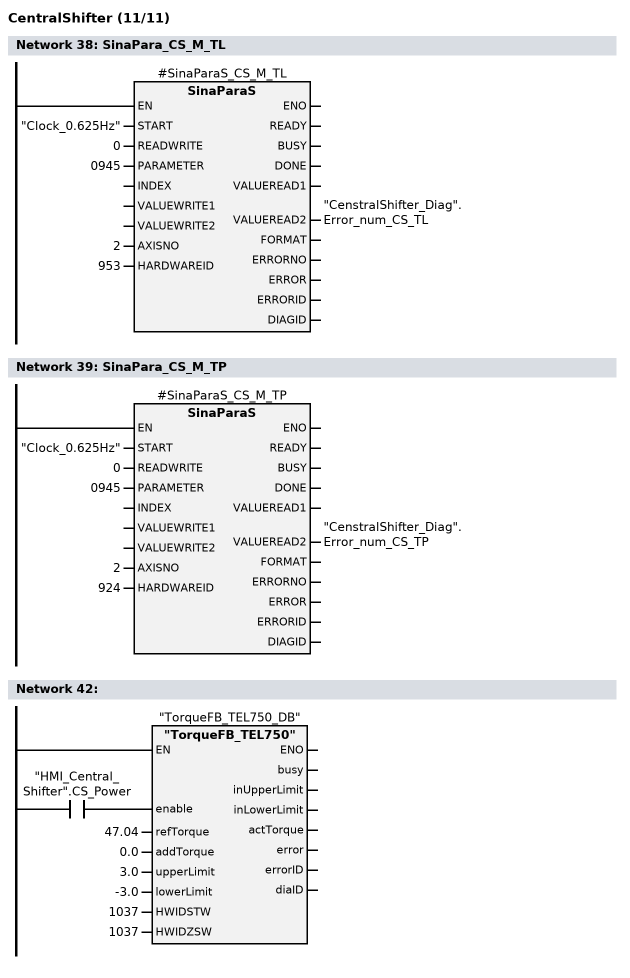
   RUNG wire#powerrail
      #SinaParaS_CS_M_TL.SinaParaS(Start := "Clock_0.625Hz", ReadWrite := 0, Parameter := 0945, Index :=, ValueWrite1 :=, ValueWrite2 :=, AxisNo := 2, hardwareId := 953, Ready =>, Busy =>, Done =>, ValueRead1 =>, ValueRead2 => "CenstralShifter_Diag".Error_num_CS_TL, Format =>, ErrorNo =>, Error =>, ErrorId =>, DiagId =>)
   END_RUNG
   // the same network as SCL:
   #SinaParaS_CS_M_TL(Start := "Clock_0.625Hz",   // SinaParaS
                      ReadWrite := 0,
                      Parameter := 0945,
                      AxisNo := 2,
                      hardwareId := 953,
                      ValueRead2 => "CenstralShifter_Diag".Error_num_CS_TL);
END_REGION

REGION Network 39: SinaPara_CS_M_TP
   RUNG wire#powerrail
      #SinaParaS_CS_M_TP.SinaParaS(Start := "Clock_0.625Hz", ReadWrite := 0, Parameter := 0945, Index :=, ValueWrite1 :=, ValueWrite2 :=, AxisNo := 2, hardwareId := 924, Ready =>, Busy =>, Done =>, ValueRead1 =>, ValueRead2 => "CenstralShifter_Diag".Error_num_CS_TP, Format =>, ErrorNo =>, Error =>, ErrorId =>, DiagId =>)
   END_RUNG
   // the same network as SCL:
   #SinaParaS_CS_M_TP(Start := "Clock_0.625Hz",   // SinaParaS
                      ReadWrite := 0,
                      Parameter := 0945,
                      AxisNo := 2,
                      hardwareId := 924,
                      ValueRead2 => "CenstralShifter_Diag".Error_num_CS_TP);
END_REGION

REGION Network 40 (SCL)
   #Active_Alarm := 0;

   IF "CenstralShifter_Diag".Error_num_CS_PL <> 0 THEN
       #Active_Alarm.%X0 := TRUE;
   END_IF;

   IF "CenstralShifter_Diag".Error_num_CS_PP <> 0 THEN
       #Active_Alarm.%X1 := TRUE;
   END_IF;

   IF "CenstralShifter_Diag".Error_num_CS_TL <> 0 THEN
       #Active_Alarm.%X2 := TRUE;
   END_IF;

   IF "CenstralShifter_Diag".Error_num_CS_TP <> 0 THEN
       #Active_Alarm.%X3 := TRUE;
   END_IF;
END_REGION

REGION Network 41 (SCL)
   (*"CS_Drive_PP_Actor_Interface_TorqueDataAddressOut".UpperTorqueLimit := 16#4000;
   "CS_Drive_PP_Actor_Interface_TorqueDataAddressOut".LowerTorqueLimit := -16#4000;

   IF #MC_MOVEJOG_CS_Virtual.JogForward THEN
       "CS_Drive_PL_Actor_Interface_TorqueDataAddressOut".UpperTorqueLimit := "CS_Drive_PP_Actor_Interface_TorqueDataAddressIn".ActualTorque;

       "CS_Drive_PL_Actor_Interface_TorqueDataAddressOut".LowerTorqueLimit := -1* "CS_Drive_PP_Actor_Interface_TorqueDataAddressIn".ActualTorque;

   ELSIF #MC_MOVEJOG_CS_Virtual.JogBackward THEN
       "CS_Drive_PL_Actor_Interface_TorqueDataAddressOut".UpperTorqueLimit := -1*"CS_Drive_PP_Actor_Interface_TorqueDataAddressIn".ActualTorque;

       "CS_Drive_PL_Actor_Interface_TorqueDataAddressOut".LowerTorqueLimit :=  "CS_Drive_PP_Actor_Interface_TorqueDataAddressIn".ActualTorque;

       ;
   ELSE
       "CS_Drive_PL_Actor_Interface_TorqueDataAddressOut".UpperTorqueLimit := 16#4000;

       "CS_Drive_PL_Actor_Interface_TorqueDataAddressOut".LowerTorqueLimit := - 16#4000;
   END_IF;
END_REGION

REGION Network 42
   RUNG wire#powerrail
      "TorqueFB_TEL750_DB"(enable := wire#w1, refTorque := 47.04, addTorque := 0.0, upperLimit := 3.0, lowerLimit := -3.0, HWIDSTW := 1037, HWIDZSW := 1037, busy =>, inUpperLimit =>, inLowerLimit =>, actTorque =>, error =>, errorID =>, diaID =>)
   END_RUNG
   RUNG wire#powerrail
      Contact( "HMI_Central_Shifter".CS_Power )
   END_RUNG wire#w1
   // the same network as SCL:
   "TorqueFB_TEL750_DB"(enable := "HMI_Central_Shifter".CS_Power,   // "TorqueFB_TEL750"
                        refTorque := 47.04,
                        addTorque := 0.0,
                        upperLimit := 3.0,
                        lowerLimit := -3.0,
                        HWIDSTW := 1037,
                        HWIDZSW := 1037);
END_REGION
END_FUNCTION_BLOCK

FUNCTION_BLOCK "CentralShifter_AutoDrive"   // FB11, LAD
{ S7_Optimized_Access := 'TRUE' }
// stored: MemoryReserve 100, SetENOAutomatically false
   VAR_INPUT
      Destination_Pos : DInt;
      Actual_Pos : DInt;
      Drive_To_Pos : Bool;
   END_VAR
   VAR_OUTPUT
      Auto_Speed : Real;
      Auto_Drive_Forward : Bool;
      Auto_Drive_Backward : Bool;
      Deceleration : Real;
   END_VAR
   VAR
      distance : DInt;
      tolerance : Real := 4.0;
      prevSpeed : Real;
      StartSpeed : Real := 380.0;
      EndSpeed : Real := 75.0;
      DecelTimer : TON_TIME;
      progress { S7_SetPoint := 'True'} : Real;
      StopRampTimer : TON_TIME;
      RampActive { S7_SetPoint := 'True'} : Bool;
      LastDirection : Int;
      StopProgress : Real;
      Vel_To_Stop : Real;
      Drive_To_Pos_Last : Bool;
      StopRampTimer_1 : TON_TIME;
      DriveOffTimer { S7_SetPoint := 'True'} : TON_TIME;
   END_VAR
BEGIN

REGION Network 1 (SCL)
   #distance := ABS(#Destination_Pos - #Actual_Pos);

   // --- wykrywanie zbocza opadającego przycisku ---
   IF NOT #Drive_To_Pos AND #Drive_To_Pos_Last THEN
       // Po puszczeniu przycisku — aktywuj rampę (jeśli jest poza tolerancją)
       IF #distance > #tolerance THEN
           #RampActive := TRUE;
           #StopRampTimer(IN := TRUE,
                          PT := T#2s); // 2 sekundy rampy
           #Vel_To_Stop := "CS_Drive_PL".Velocity; // zapamiętaj prędkość do wyhamowania
       ELSE
           // Jeśli już w tolerancji — od razu stop
           #RampActive := FALSE;
           #StopRampTimer.IN :=0;
           #Auto_Speed := 0.0;
           #Auto_Drive_Forward := FALSE;
           #Auto_Drive_Backward := FALSE;
       END_IF;
   END_IF;

   #Drive_To_Pos_Last := #Drive_To_Pos;

   // --- Główna logika ruchu ---
   IF #Drive_To_Pos THEN
       // --- Tryb aktywnego ruchu ---
       IF #distance <= #tolerance THEN
           "HMI_Central_Shifter".CS_Status_Auto_Go_to_Des := 2;
           #Auto_Drive_Forward := FALSE;
           #Auto_Drive_Backward := FALSE;
           #Auto_Speed := 0.0;
           #DecelTimer.IN := FALSE;
       ELSE
           "HMI_Central_Shifter".CS_Status_Auto_Go_to_Des := 1;

           // Kierunek
           IF #Actual_Pos > #Destination_Pos THEN
               #Auto_Drive_Forward := TRUE;
               #Auto_Drive_Backward := FALSE;
               #LastDirection := 1;
           ELSE
               #Auto_Drive_Forward := FALSE;
               #Auto_Drive_Backward := TRUE;
               #LastDirection := -1;
           END_IF;

           // Rampowanie w zależności od odległości
           IF #distance > 5000.0 THEN
               #Auto_Speed := #StartSpeed;
               #DecelTimer.IN := FALSE;
           ELSE
               #DecelTimer(IN := TRUE,
                           PT := T#5s);
               #progress := (5000.0 - #distance) / 5000.0;
               IF #progress > 1.0 THEN
                   #progress := 1.0;
               END_IF;
               #Auto_Speed := #StartSpeed - #progress * (#StartSpeed - #EndSpeed);
           END_IF;
       END_IF;

       // Reset rampy podczas aktywnego ruchu
       #RampActive := FALSE;
       #StopRampTimer.IN := FALSE;

   ELSE
       // --- Tryb hamowania rampą po puszczeniu przycisku ---
       IF #RampActive THEN
           #StopProgress := INT_TO_REAL(TIME_TO_INT(#StopRampTimer.ET)) / INT_TO_REAL(TIME_TO_INT(T#2s));
           IF #StopProgress > 1.0 THEN
               #StopProgress := 1.0;
           END_IF;

           // Liniowe zmniejszanie prędkości
           #Auto_Speed := (1.0 - #StopProgress) * #Vel_To_Stop;

           // Kierunek zgodny z ostatnim
           IF #LastDirection = 1 THEN
               #Auto_Drive_Forward := TRUE;
               #Auto_Drive_Backward := FALSE;
           ELSIF #LastDirection = -1 THEN
               #Auto_Drive_Forward := FALSE;
               #Auto_Drive_Backward := TRUE;
           ELSE
               #Auto_Drive_Forward := FALSE;
               #Auto_Drive_Backward := FALSE;
           END_IF;

           // Po zakończeniu rampy
           IF #StopRampTimer.Q THEN
               #Auto_Speed := 0.0;
               #Auto_Drive_Forward := FALSE;
               #Auto_Drive_Backward := FALSE;
               #RampActive := FALSE;
               #StopRampTimer.IN :=0;
               #LastDirection := 0;
           END_IF;
       ELSE
           // Jeśli rampa nieaktywna — wymuszone zatrzymanie
           #Auto_Speed := 0.0;
           #Auto_Drive_Forward := FALSE;
           #Auto_Drive_Backward := FALSE;
           #StopRampTimer.IN := FALSE;
       END_IF;
   END_IF;

